# B&R Automation Studio project x20ost (part 5)

#### bnrsmartsensor.c
```c
/********************************************************************
 * COPYRIGHT -- Kontora
 ********************************************************************
 * Program: bnrmain
 * File: bnrlsens.c
 * Author: Abramenya
 * Created: January 19, 2009
 *******************************************************************/

#include "bnrsmartsensor.h"
#if MYSYSTEM_ID != 5
#ifdef _DEFAULT_INCLUDES
 #include <AsDefault.h>
#endif
extern BYTE *chSensType[];
extern BYTE *chParType[];
#ifdef WIN32
void LCPIDpara(LCPIDpara_typ *pPara){}
void LCPID(LCPID_typ *pPid){};
void LCCounter(LCCounter_typ *pCounder){};
#endif
_GLOBAL LCPIDpara_typ lParaTyp;
void CSmartSensor_InitSensor(This,PVOID pvParam)
{
    DECLARE_MULTI_OPEN(CSmartSensor,CSensor)
	SNSPARAMTABLE *pParam = (SNSPARAMTABLE*)pvParam;
	COutGate *pG = pB->m_pOutGate[0];
    pT->SetState(pT,TRUE);
	pT->m_wExtError = 0;
	pT->m_sSNSParam.enable    = pT->GetState(pT);
	pT->m_sSNSParam.enter     = pT->GetState(pT);
	pT->m_sSNSParam.Y_min     = (UINT)(pG->m_rMinRamp*pB->m_sPT.m_swMaxAcpOut);
	pT->m_sSNSParam.Y_max     = (UINT)(pG->m_rMaxRamp*pB->m_sPT.m_swMaxAcpOut);
	pT->m_sSNSParam.dY_max    = pB->m_sPT.m_rlDy;
	pT->m_sSNSParam.Kp        = pB->m_sPT.m_rlKp;
	pT->m_sSNSParam.Tn        = pB->m_sPT.m_rlTn;
	pT->m_sSNSParam.Tv        = pB->m_sPT.m_rlTv;
	pT->m_sSNSParam.Tf        = pB->m_sPT.m_rlTf;
	pT->m_sSNSParam.Kw        = pB->m_sPT.m_rlKw;
	pT->m_sSNSParam.Kfbk      = pB->m_sPT.m_rlKfbk;
	pT->m_sSNSParam.fbk_mode  = LCPID_FBK_MODE_INTERN;
	if (pB->m_sPT.m_swPidDiffMode==0)pT->m_sSNSParam.d_mode = LCPID_D_MODE_X;
	if (pB->m_sPT.m_swPidDiffMode==1)pT->m_sSNSParam.d_mode = LCPID_D_MODE_E;
	pT->m_sSNSParam.calc_mode = LCPID_CALC_MODE_FAST;
	LCPIDpara(&pT->m_sSNSParam);
	pT->m_sLCPid.enable       = pT->GetState(pT);
	pT->m_sLCPid.A            = pB->m_sPT.m_rlA;//500;
	pT->m_sLCPid.Y_man	      = pB->m_sPT.m_rlYman;
	pT->m_sLCPid.Y_fbk        = 0;
	pB->m_nInPin              = pB->m_nIniValue;
	pT->m_sLCPid.X            = pB->m_nInPin;
	pT->m_sLCPid.W            = pB->m_iPHiLimit;
	pT->m_sLCPid.Y            = pB->m_pOutGate[0]->m_wCurrOpenState;
	pB->m_nOutPin             = 0;
	pT->m_sLCPid.e            = 0;
	pT->m_sLCPid.Yi           = 0;
	pT->m_sLCPid.Yp           = 0;
	pT->m_sLCPid.Yd           = 0;
	pT->m_sLCPid.hold_I       = 0;
	if (pB->m_sPT.m_sbyMode==SNS_MD_MANU)pT->SetMode(pT,LCPID_OUT_MODE_MAN);
	if (pB->m_sPT.m_sbyMode==SNS_MD_AUTO)pT->SetMode(pT,LCPID_OUT_MODE_AUTO);
    pT->m_sLCPid.ident        = pT->m_sSNSParam.ident;
	LCPID(&pT->m_sLCPid);
	#ifdef DEB_CSmartSensor
	Info("\n(%b)CISNS::>Create SNS.:%s.:%s.Rng:[%w..%w].AlarmRng:[%w..%w]",
		&pB->m_bySensorID,
		chSensType[pB->m_bySensorType],
		chParType[pB->m_byParamType],
		&pB->m_iLoLimit,&pB->m_iHiLimit,
		&pB->m_iLoAlmLimit,&pB->m_iHiAlmLimit
	);
	#endif
}
void CSmartSensor_IncInput(This,INT16 wParam)
{
    DECLARE_MULTI_OPEN(CSmartSensor,CSensor)
    pT->m_wExtError += wParam;
	//Info("\n(%b)CSMSN::>DC(%b,%b)PR_INC::%w.",&pB->m_bySystemID,&pB->m_byDirection,&pB->m_bySensorID,&pB->m_nInPin);
}
void CSmartSensor_SetInput(This,SPIN *pValue)
{
    DECLARE_MULTI_OPEN(CSmartSensor,CSensor)
	pB->m_nInPin = pValue->iValue;
    //Info("\n(%b)CSMSN::>DC(%b,%b)PR_X::%w.",&pB->m_bySystemID,&pB->m_byDirection,&pB->m_bySensorID,&pB->m_nInPin);
}
void CSmartSensor_SetOutput(This,BYTE byNumber,SPIN *pValue)
{
	DECLARE_MULTI_OPEN(CSmartSensor,CSensor)
	COutGate *pG0 = pB->m_pOutGate[byNumber];
	pB->m_nOutPin = pValue->iValue;
	if(pG0)pG0->SetGate(pG0,pB->m_nOutPin);
}
void CSmartSensor_PreProc(This)
{
    DECLARE_MULTI_OPEN(CSmartSensor,CSensor)
	CInputGate *pI = pB->m_nInp;
	if(pB->m_byPidMode==SDIR)pB->m_nInPin = pI->GetInput(pI); else
	if(pB->m_byPidMode==SINV)pB->m_nInPin = pB->m_nAcpMax-pI->GetInput(pI);
	if(pB->m_sPT.m_sbyMode==SNS_MD_LOOP) pB->m_nInPin += pT->m_wExtError;
}
_GLOBAL LCPID_typ lPtyp;
void CSmartSensor_Processing(This)
{
    DECLARE_MULTI_OPEN(CSmartSensor,CSensor)
    #ifndef WIN32
	#ifdef MY_MODEL
	REAL rRes,rOut;
	#endif
	LCCounter(&pT->m_sCounter);
	pT->m_sLCPid.W        = pB->m_iPHiLimit;
	pT->m_sLCPid.X        = pB->m_nInPin;
	pT->m_sLCPid.basetime = pT->m_sCounter.mscnt;
	LCPID(&pT->m_sLCPid);
	#ifdef MY_MODEL
	rOut = (REAL)pT->m_sLCPid.Y;
	rRes = (rOut/378.0)-2.0;
	if((pB->m_nInPin+(INT16)rRes)>32760)pB->m_nInPin = 32760;else
	if((pB->m_nInPin+(INT16)rRes)<0)pB->m_nInPin = 0;else
	pB->m_nInPin += (INT16)rRes;
	#endif
	pB->m_nOutPin = pT->m_sLCPid.Y;
    #else
	pT->m_sLCPid.W   = pB->m_iPHiLimit;
  	pT->m_sLCPid.X   = pB->m_nInPin;
	pB->m_nOutPin    = pT->m_sLCPid.Y;
    #endif
	//pB->AddStatData(pB,pT->m_sLCPid.Y,pT->m_sLCPid.Yi,pT->m_sLCPid.Yp);
}
void CSmartSensor_PostProc(This)
{
    DECLARE_MULTI_OPEN(CSmartSensor,CSensor)
	COutGate *pG0 = pB->m_pOutGate[0];
    if(pG0)pG0->SetGate(pG0,pB->m_nOutPin);
}
void CSmartSensor_Serialize(This,BOOL byDir)
{
	DECLARE_MULTI_OPEN(CSmartSensor,CSensor)
	COutGate *pG0 = pB->m_pOutGate[0];
	if (byDir==TRUE)if(pG0)pG0->SetGate(pG0,pB->m_nOutPin);
	if (byDir==FALSE)
	{
	 pT->m_sLCPid.Y = pG0->m_wCurrOpenState;
	 pG0->StopGate(pG0);
	}
}
void CSmartSensor_RunAutomat(This)
{
    DECLARE_MULTI_OPEN(CSmartSensor,CSensor)
	BYTE i;
	COutGate *pG;
	if(pB->m_dwAutoTime++%5==0)
	{
	 pB->EventGen(pB);
	 for (i=0;i<pB->m_byAmOutGate;i++){pG = pB->m_pOutGate[i];pG->RunGate(pG);}
	}
}
void CSmartSensor_CaptureData(This)
{
	DECLARE_MULTI_OPEN(CSmartSensor,CSensor)
	COutGate *pG0 = pB->m_pOutGate[0];
    pB->OpenGate(pB);
	pB->AddData(pB,(DINT)pB->m_nInPin);
	pB->AddData(pB,(DINT)pT->m_sLCPid.W);
	pB->AddData(pB,(DINT)(pG0->GetGate(pG0)));
	pB->AddData(pB,pT->m_sLCPid.e);
	pB->AddData(pB,pT->m_sLCPid.Yi);
	pB->AddData(pB,pT->m_sLCPid.Yp);
	pB->AddData(pB,pT->m_sLCPid.Yd);
	pB->CloseGate(pB);
}
USINT CSmartSensor_GetMode(This)
{
    DECLARE_MULTI_OPEN(CSmartSensor,CSensor)
	return pT->m_sLCPid.out_mode;
}
void CSmartSensor_SetMode(This,USINT uMode)
{
    DECLARE_MULTI_OPEN(CSmartSensor,CSensor)
	pT->m_sLCPid.out_mode = uMode;
}
BOOL CSmartSensor_GetState(This)
{
    DECLARE_MULTI_OPEN(CSmartSensor,CSensor)
	return pT->m_blState;
}
void CSmartSensor_SetState(This,BOOL blBool)
{
    DECLARE_MULTI_OPEN(CSmartSensor,CSensor)
	pT->m_sSNSParam.enable    = blBool;
	pT->m_sSNSParam.enter     = blBool;
	pT->m_sLCPid.enable       = blBool;
	pT->m_blState             = blBool;
	LCPIDpara(&pT->m_sSNSParam);
}
//_GLOBAL REAL rKP;
//_GLOBAL INT  i16Param;
void CSmartSensor_EventHandler(This,SMESSAGE *pMsg)
{
    DECLARE_MULTI_OPEN(CSmartSensor,CSensor)
	SPIN nPin;
	REAL rlParam;
	INT16 wParam;
	BYTE byLen,byInitType,byPType,byPLen,*pR=(BYTE*)&rlParam;
	switch(pMsg->m_sbyType)
	{
      case EV_SMSNS_SET_PARAM_REQ:
		   byLen      = pMsg->m_sbyInfo[0];
		   byInitType = pMsg->m_sbyInfo[1];
		   byPType    = pMsg->m_sbyInfo[2];
		   byPLen     = pMsg->m_sbyInfo[3];
           #ifdef DEB_CSmartSensor
 		   //Info("\n(%b)CSMSN::>DC(%b,%b)SSP:%M.",&pB->m_bySystemID,&pB->m_byDirection,&pB->m_bySensorID,(BYTE*)pMsg);
           #endif
		   if(byInitType==SNS_SENS_OUT)
		   {
			 switch(byPType)
			 {
			  case PR_OMIN:
				   rlParam = pB->GetRealParam(pT,&pMsg->m_sbyInfo[4]);
				   pT->m_sSNSParam.Y_min = (UINT)(rlParam*pB->m_sPT.m_swMaxAcpOut);
				   LCPIDpara(&pT->m_sSNSParam);
			  break;
			  case PR_OMAX:
				   rlParam = pB->GetRealParam(pB,&pMsg->m_sbyInfo[4]);
				   pT->m_sSNSParam.Y_max = (UINT)(rlParam*pB->m_sPT.m_swMaxAcpOut);
				   LCPIDpara(&pT->m_sSNSParam);
			  break;
			  default:
			  break;
			 }
		   }
		   if(byInitType==SNS_PARA_INI)
		   {
		    switch(byPType)
			{
			 case PR_Y_max:
				  pT->m_sSNSParam.Y_max  = pB->GetWordParam(pB,&pMsg->m_sbyInfo[4]);
				  pB->m_sGT.wHiLimit     = pT->m_sSNSParam.Y_max;
                  pB->m_pOutGate[0]->SetHiLimit(pB->m_pOutGate[0],pB->m_sGT.wHiLimit);
			 break;
			 case PR_Y_min:
				  pT->m_sSNSParam.Y_min  = pB->GetWordParam(pB,&pMsg->m_sbyInfo[4]);
			 break;
			 case PR_dY_max:
				  pT->m_sSNSParam.dY_max = pB->GetRealParam(pB,&pMsg->m_sbyInfo[4]);
				  pB->m_sPT.m_rlDy       = pT->m_sSNSParam.dY_max;
			 break;
			 case PR_Kp:
				  pT->m_sSNSParam.Kp     = pB->GetRealParam(pB,&pMsg->m_sbyInfo[4]);
				  pB->m_sPT.m_rlKp       = pT->m_sSNSParam.Kp;
			 break;
			 case PR_Tn:
				  pT->m_sSNSParam.Tn     = pB->GetRealParam(pB,&pMsg->m_sbyInfo[4]);
				  pB->m_sPT.m_rlTn       = pT->m_sSNSParam.Tn;
			 break;
			 case PR_Tv:
				  pT->m_sSNSParam.Tv     = pB->GetRealParam(pB,&pMsg->m_sbyInfo[4]);
				  pB->m_sPT.m_rlTv       = pT->m_sSNSParam.Tv;
			 break;
			 case PR_Tf:
				  pT->m_sSNSParam.Tf     = pB->GetRealParam(pB,&pMsg->m_sbyInfo[4]);
				  pB->m_sPT.m_rlTf       = pT->m_sSNSParam.Tf;
			 break;
			 case PR_Kw:
				  pT->m_sSNSParam.Kw     = pB->GetRealParam(pB,&pMsg->m_sbyInfo[4]);
				  pB->m_sPT.m_rlKw       = pT->m_sSNSParam.Kw;
			 break;
			 case PR_Kfbk:
				  pT->m_sSNSParam.Kfbk   = pB->GetRealParam(pB,&pMsg->m_sbyInfo[4]);
				  pB->m_sPT.m_rlKfbk     = pT->m_sSNSParam.Kfbk;
			 break;
			 case PR_PrEn:
				  pB->m_sPT.m_swPidDiffMode = 0;
				  pT->m_sSNSParam.enable = (BOOL)pMsg->m_sbyInfo[4];
				  pB->m_sPT.m_swPidDiffMode = pT->m_sSNSParam.enable;
				  if (pB->m_sPT.m_swPidDiffMode==0)pT->m_sSNSParam.d_mode = LCPID_D_MODE_X;
				  if (pB->m_sPT.m_swPidDiffMode==1)pT->m_sSNSParam.d_mode = LCPID_D_MODE_E;
				  #ifdef DEB_CSmartSensor
				  Info("\n(%b)CSMSN::>DC(%b,%b)PR_PrEn.",&pB->m_bySystemID,&pB->m_byDirection,&pB->m_bySensorID);
				  #endif
			 break;
			 default:
			 break;
			}
		    LCPIDpara(&pT->m_sSNSParam);
		   }
		   if((byInitType==SNS_PIDC_INI)||(byInitType==SNS_SENS_INI))
		   {
			switch(byPType)
			{
			 case PR_W:
				  wParam = pB->GetWordParam(pB,&pMsg->m_sbyInfo[4]);
				  if(pB->m_byPidMode==SINV) wParam = pB->m_nAcpMax-wParam;
				  pB->m_sPT.m_swHiOper = pB->AcpToReal(pB,wParam);
   			      pT->m_sLCPid.W = wParam;
				  pB->SetHiLimit(pB,wParam);
			 break;
			 case PR_X:
				  nPin.iValue = pB->GetWordParam(pB,&pMsg->m_sbyInfo[4]);
				  pT->m_sLCPid.X = nPin.iValue;
    			  pT->SetInput(pT,&nPin);
			 break;
			 case PR_A:
				  pT->m_sLCPid.A  = pB->GetWordParam(pB,&pMsg->m_sbyInfo[4]);
				  pB->m_sPT.m_rlA = pT->m_sLCPid.A;
			 break;
			 case PR_Y_man:
				  pT->m_sLCPid.Y_man = pB->GetWordParam(pB,&pMsg->m_sbyInfo[4]);
				  pB->m_sPT.m_rlYman = pT->m_sLCPid.Y_man;
			 break;
			 case PR_out_mode:
			      if(pMsg->m_sbyInfo[4]==0)
				  {
				   #ifdef DEB_CSmartSensor
				   Info("\n(%b)CSMSN::>DC(%b,%b)SNS_MD_MANU.",&pB->m_bySystemID,&pB->m_byDirection,&pB->m_bySensorID);
				   #endif
				  }
			      if(pMsg->m_sbyInfo[4]==1)
				  {
				   pT->m_sLCPid.out_mode = LCPID_OUT_MODE_AUTO;
				   #ifdef DEB_CSmartSensor
				   Info("\n(%b)CSMSN::>DC(%b,%b)SNS_MD_AUTO.",&pB->m_bySystemID,&pB->m_byDirection,&pB->m_bySensorID);
				   #endif
				  }
			      if(pMsg->m_sbyInfo[4]==2)
				  {
				   pT->m_sLCPid.out_mode = LCPID_OUT_MODE_AUTO;
				   #ifdef DEB_CSmartSensor
				   Info("\n(%b)CSMSN::>DC(%b,%b)SNS_MD_LOOP.",&pB->m_bySystemID,&pB->m_byDirection,&pB->m_bySensorID);
				   #endif
				  }
			 break;
			 case PR_PidEn:
				  pT->m_sLCPid.enable   = (BOOL)pMsg->m_sbyInfo[4];
				  #ifdef DEB_CSmartSensor
				  Info("\n(%b)CSMSN::>DC(%b,%b)PR_PidEn.",&pB->m_bySystemID,&pB->m_byDirection,&pB->m_bySensorID);
				  #endif
			 break;
			 default:
			 break;
			}
			LCPID(&pT->m_sLCPid);
		   }
  	  break;
	  default:
	  break;
	};
}
void CSmartSensor_GetParam(This,BYTE byOwner)
{
    DECLARE_MULTI_OPEN(CSmartSensor,CSensor)
	SHMESSAGE m_sMsg;
	BYTE *pP = &m_sMsg.m_sbyInfo[1];
	SPIDPARAM sP;
	INT nSS = sizeof(SPIDPARAM);
    m_sMsg.m_sbyFrom      = MDL_DIRMD;
    m_sMsg.m_sbyFor       = byOwner;
    m_sMsg.m_sbyIntType   = DEV_ARM_PORT_TCP;
    m_sMsg.m_sbyType      = EV_SENSR_GET_PDPARAM_IND;
    m_sMsg.m_sbyServerID  = pB->m_bySystemID;
    m_sMsg.m_sbyDirection = pB->m_byDirection;
	m_sMsg.m_sbySensor  = pB->m_bySensorID;
    sP.Kp     = pB->GetRealParam(pB,(BYTE*)&pT->m_sSNSParam.Kp);
    sP.Tn     = pB->GetRealParam(pB,(BYTE*)&pT->m_sSNSParam.Tn);
    sP.Tv     = pB->GetRealParam(pB,(BYTE*)&pT->m_sSNSParam.Tv);
    sP.Tf     = pB->GetRealParam(pB,(BYTE*)&pT->m_sSNSParam.Tf);
    sP.Kw     = pB->GetRealParam(pB,(BYTE*)&pT->m_sSNSParam.Kw);
	sP.Kfbk   = pB->GetRealParam(pB,(BYTE*)&pT->m_sSNSParam.Kfbk);
	sP.Y_max  = pB->GetWordParam(pB,(BYTE*)&pT->m_sSNSParam.Y_max);
    sP.Y_min  = pB->GetWordParam(pB,(BYTE*)&pT->m_sSNSParam.Y_min);
    sP.dY_max = pB->GetRealParam(pB,(BYTE*)&pT->m_sSNSParam.dY_max);
    sP.enable = (BYTE)pT->m_sSNSParam.enable;
	pT->m_sLCPid.W = pB->m_iPHiLimit;
	sP.W      = pB->GetWordParam(pB,(BYTE*)&pT->m_sLCPid.W);
	sP.X      = pB->GetWordParam(pB,(BYTE*)&pT->m_sLCPid.X);
	sP.A      = pB->GetWordParam(pB,(BYTE*)&pT->m_sLCPid.A);
	sP.Y_man  = pB->GetWordParam(pB,(BYTE*)&pT->m_sLCPid.Y_man);
    if(pT->m_sLCPid.out_mode == LCPID_OUT_MODE_MAN) sP.out_mode = 0;
	if(pT->m_sLCPid.out_mode == LCPID_OUT_MODE_AUTO)sP.out_mode = 1;
	sP.enabled = (BYTE)pT->m_sLCPid.enable;
	m_sMsg.m_sbyInfo[0] = 1+ sizeof(SPIDPARAM);
	memcpy(&m_sMsg.m_sbyInfo[1],&sP,sizeof(SPIDPARAM));
    m_sMsg.m_swLen = 9 + m_sMsg.m_sbyInfo[0];
	#ifdef DEB_CSmartSensor
	Info("\n(%b)CSMSN::>DC(%b,%b)SFF:%M.",&pB->m_bySystemID,&pB->m_byDirection,&pB->m_bySensorID,(BYTE*)&m_sMsg);
	#endif
    FPUT(DEV_ARMOT_BOX_ID,(BYTE*)&m_sMsg.m_swLen);
}
DWORD CSmartSensor_MotToInt(This,DWORD dwData)
{
    DECLARE_MULTI_OPEN(CSmartSensor,CSensor)
	DWORD dwValue;
	BYTE *pTR = (BYTE*)&dwValue;
	BYTE *pSR = (BYTE*)&dwData;
    #ifndef WIN32
	pTR[3] = pSR[0];
	pTR[2] = pSR[1];
	pTR[1] = pSR[2];
	pTR[0] = pSR[3];
    #else
	memcpy(pTR,pSR,4);
    #endif
	return dwValue;
}
void CSmartSensor_CSmartSensor(This)
{
    DECLARE_MULTI_OPEN(CSmartSensor,CSensor)
	DECLARE_REGISTRATION(CSmartSensor,SetMode)
	DECLARE_REGISTRATION(CSmartSensor,SetState)
	DECLARE_REGISTRATION(CSmartSensor,GetState)
	DECLARE_REGISTRATION(CSmartSensor,MotToInt)
	DECLARE_VIRTUAL_FUNC(CSmartSensor,EventHandler)
	DECLARE_VIRTUAL_FUNC(CSmartSensor,SetInput)
	DECLARE_VIRTUAL_FUNC(CSmartSensor,SetOutput)
	DECLARE_VIRTUAL_FUNC(CSmartSensor,InitSensor)
	DECLARE_VIRTUAL_FUNC(CSmartSensor,PreProc)
	DECLARE_VIRTUAL_FUNC(CSmartSensor,Processing)
	DECLARE_VIRTUAL_FUNC(CSmartSensor,PostProc)
	DECLARE_VIRTUAL_FUNC(CSmartSensor,CaptureData)
	DECLARE_VIRTUAL_FUNC(CSmartSensor,GetParam)
	DECLARE_VIRTUAL_FUNC(CSmartSensor,IncInput)
	DECLARE_VIRTUAL_FUNC(CSmartSensor,RunAutomat)
	DECLARE_VIRTUAL_FUNC(CSmartSensor,Serialize)
}
void CSmartSensor_DCSmartSensor(This)
{
	DECLARE_MULTI_OPEN(CSmartSensor,CSensor)
	DestroyObjectB(CSensor,pB);
}
DECLARE_MULTI_CREATE(CSmartSensor,CSensor)
#endif
```

#### bnrsystemtimer.c
```c
/********************************************************************
 * COPYRIGHT -- Kontora
 ********************************************************************
 * Program: bnrmain
 * File: bnrlsens.c
 * Author: Abramenya
 * Created: January 19, 2009
 *******************************************************************/

#include "bnrsystemtimer.h"
#ifdef _DEFAULT_INCLUDES
 #include <AsDefault.h>
#endif
void CSystemTimer_RunTimer(This)
{
     DECLARE_SINGLE_OPEN(CSystemTimer)
	 if(pT->m_blTimerState==TRUE)
	 {
	  //Info("\nTime[%w]",&pT->m_dwTime);
      if (pT->m_dwTime--==0)
	  {
		 //Info("\nTime[%w]",&pT->m_dwTime);
         pT->DoAction(pC);
		 pT->m_dwTime = 0;
		 pT->m_blTimerState = FALSE;
		 return;
	  }
	 }
}
void CSystemTimer_DoAction(This)
{
     DECLARE_SINGLE_OPEN(CSystemTimer)
}
void CSystemTimer_OfTimer(This)
{
     DECLARE_SINGLE_OPEN(CSystemTimer)
	 pT->m_blTimerState = FALSE;
     pT->m_dwTime = 0;
}
void CSystemTimer_OnTimer(This,DWORD dwTime)
{
     DECLARE_SINGLE_OPEN(CSystemTimer)
	 pT->m_blTimerState = TRUE;
     pT->m_dwTime = dwTime;
}
void CSystemTimer_SetTimerID(This,BYTE byTimerID)
{
     DECLARE_SINGLE_OPEN(CSystemTimer)
	 pT->m_byTimerID = byTimerID;
}
void CSystemTimer_CSystemTimer(This)
{
     DECLARE_SINGLE_OPEN(CSystemTimer)
	 DECLARE_REGISTRATION(CSystemTimer,RunTimer)
	 DECLARE_REGISTRATION(CSystemTimer,OnTimer)
	 DECLARE_REGISTRATION(CSystemTimer,OfTimer)
	 DECLARE_REGISTRATION(CSystemTimer,DoAction)
	 DECLARE_REGISTRATION(CSystemTimer,SetTimerID)
	 pT->m_dwTime = 0;
	 pT->m_blTimerState = FALSE;
	 FCTIMER(pT);
}
void CSystemTimer_DCSystemTimer(This)
{
	 DECLARE_SINGLE_OPEN(CSystemTimer)
	 FDTIMER(pT);
}
DECLARE_SINGLE_CREATE(CSystemTimer)
```

#### bnrtelecontrol.c
```c
/********************************************************************
 * COPYRIGHT -- Kontora
 ********************************************************************
 * Program: bnrmain
 * File: bnrlsens.c
 * Author: Abramenya
 * Created: January 19, 2009
 *******************************************************************/

#include "bnrtelecontrol.h"
#ifdef _DEFAULT_INCLUDES
#include <AsDefault.h>
#endif
void CTeleControl_InitTCHN(This,PVOID psTable)
{
    DECLARE_MULTI_OPEN(CTeleControl,CTeleSensor)
	//BYTE i;
	pT->pP       = (STUPARAM*)psTable;
	pT->m_pbOT   = (BOOL*)pB->m_pvValue;
	pB->m_byType = REG_SOFTU_ADDR;
	pT->m_byStPulce  = FALSE;
	//pB->SaveChange(pB,EV_INI_CH,*pT->m_pbOT);
	//for(i=0;i<5;i++) pB->SaveChange(pB,EV_1T0_CH,i);
	//pT->m_bySetPulce = pT->pP->byCSetPulce;
    #ifdef DEB_CTeleControl
	//Info("\n(%b)CTLCT::>Create CTeleControl.",&pB->m_byID);
    #endif
}
void CTeleControl_PreProc(This)
{
    DECLARE_MULTI_OPEN(CTeleControl,CTeleSensor)
}
_GLOBAL INT nTCCH;
void CTeleControl_Processing(This)
{
	DECLARE_MULTI_OPEN(CTeleControl,CTeleSensor)
	if (pB->m_byID==5)	nTCCH++;
	if(pT->pP->byState==EN_OPEN)
	{
	 if(pT->m_byStPulce==TRUE)
	 {
	 if (--pT->m_bySetPulce==0)
	 {
	   if(*pT->m_pbOT==FALSE)
	   {
	   *pT->m_pbOT = TRUE;
	   pB->SaveChange(pB,EV_0T1_ST,1,FALSE);
	   }else
	   if(*pT->m_pbOT==TRUE )
	   {
	   *pT->m_pbOT = FALSE;
	   pB->SaveChange(pB,EV_1T0_ST,0,FALSE);
	   }
       #ifdef DEB_CTeleControl
	   Info("\n(%b)CTLCT::>SetPulce::STOP.",&pB->m_byID);
       #endif
	   pT->m_byStPulce  = FALSE;
	 }
	 }
	 pT->pP->byParam = *pT->m_pbOT;
	}
}
void CTeleControl_PostProc(This)
{
	DECLARE_MULTI_OPEN(CTeleControl,CTeleSensor)
}
void CTeleControl_SetPulce(This)
{
    DECLARE_MULTI_OPEN(CTeleControl,CTeleSensor)
	if(pT->pP->byState==EN_OPEN)
	{
	 pT->m_bySetPulce = pT->pP->byCSetPulce;
	 pT->m_byStPulce  = TRUE;
	 if (pT->pP->byPulceType==EN_DIRECT)
	 {
	  *pT->m_pbOT = TRUE;
	  pB->SaveChange(pB,EV_0T1_ST,1,FALSE);
	 }
	 if (pT->pP->byPulceType==EN_INVERT)
	 {
	  *pT->m_pbOT = FALSE;
	  pB->SaveChange(pB,EV_1T0_ST,0,FALSE);
	 }
	 #ifdef DEB_CTeleControl
	 Info("\n(%b)CTLCT::>SetPulce::START.",&pB->m_byID);
     #endif
	}
}
void CTeleControl_SetInPinEvent(This)
{
    DECLARE_MULTI_OPEN(CTeleControl,CTeleSensor)
	pB->SavePinState(pB,EV_INI_CH,*pT->m_pbOT);
}
void CTeleControl_SaveAlarmPin(This)
{
	DECLARE_MULTI_OPEN(CTeleControl,CTeleSensor)
	pB->SavePinState(pB,EV_ALP_CH,(WORD)pT->pP->byAlmState);
}
void CTeleControl_SendObsrveMsg(This)
{
    DECLARE_MULTI_OPEN(CTeleControl,CTeleSensor)
    SKPEVENT sEV;
	sEV.wLen    = sizeof(SKPEVENT);
	sEV.byType  = pB->m_byType;
    sEV.byCause = EV_CHK_CH;
	sEV.byAddr  = pB->m_byID;
	sEV.wValue  = (WORD)*pT->m_pbOT;
	GetCurTime(&sEV.sTime);
    pB->SendBroadcast(pB,&sEV);
}
BOOL CTeleControl_EventHandler(This,SMESSAGE *pMsg)
{
    DECLARE_MULTI_OPEN(CTeleControl,CTeleSensor)
	BYTE byParamType = pMsg->m_sbyInfo[3];
    #ifdef DEB_CTeleControl
	Info("\n(%b)CTLCT::>INPT::%M",&pB->m_byID,pMsg);
    #endif
	switch(pMsg->m_sbyFor)
	{
	  case DIR_101TOKP:
		   switch(pMsg->m_sbyType)
		   {
		    case PL_DATA_IND:
				 switch(byParamType)
				 {
				   case EN_STT_PULCE:
					    pT->SetPulce(pT);
				   break;
				   case EN_STT_SIGN:
					   //pT->SetPulce(pT,pT->pP->byPulceType);
				   break;
				   default:
				   break;
				 }

		    break;
			default:
            break;
		   }
      break;
	  case DIR_101MD:
	  break;
	  default:
	  break;
	}
	return TRUE;
}
void CTeleControl_CTeleControl(This)
{
    DECLARE_MULTI_OPEN(CTeleControl,CTeleSensor)
	DECLARE_REGISTRATION(CTeleControl,SetPulce)
	DECLARE_VIRTUAL_FUNC(CTeleControl,SetInPinEvent)
	DECLARE_VIRTUAL_FUNC(CTeleControl,InitTCHN)
	DECLARE_VIRTUAL_FUNC(CTeleControl,PreProc)
	DECLARE_VIRTUAL_FUNC(CTeleControl,Processing)
	DECLARE_VIRTUAL_FUNC(CTeleControl,PostProc)
	DECLARE_VIRTUAL_FUNC(CTeleControl,EventHandler)
	DECLARE_VIRTUAL_FUNC(CTeleControl,SaveAlarmPin)
	DECLARE_VIRTUAL_FUNC(CTeleControl,SendObsrveMsg)
}
void CTeleControl_DCTeleControl(This)
{
	DECLARE_MULTI_OPEN(CTeleControl,CTeleSensor)
}
DECLARE_MULTI_CREATE(CTeleControl,CTeleSensor)
```

#### bnrteleind.c
```c
/********************************************************************
 * COPYRIGHT -- Kontora
 ********************************************************************
 * Program: bnrmain
 * File: bnrlsens.c
 * Author: Abramenya
 * Created: January 19, 2009
 *******************************************************************/

#include "bnrteleind.h"
#include "bnrmain.h"
#ifdef _DEFAULT_INCLUDES
#include <AsDefault.h>
#endif
extern UINT *uipValueAI2[];
void CTeleInd_InitTCHN(This,PVOID psTable)
{
    DECLARE_MULTI_OPEN(CTeleInd,CTeleSensor)
	//BYTE i;
	pT->pP = (STIPARAM*)psTable;
	pT->m_pnIN = (WORD*)pB->m_pvValue;

	pT->m_byRemTimer   = pT->pP->byDrTimer;
	pT->m_blTmRemState = FALSE;

	pT->m_bySetTimer   = pT->pP->byDrTimer;
	pT->m_blTmSetState = FALSE;

	pT->m_blChState    = pT->pP->byDrTimer;
	pT->m_byChTimer    = FALSE;

	pT->m_byErEventCh  = EV_CHG_PR;
	pT->m_byErEventHi  = EV_CHG_PR;
	pT->m_byErEventLo  = EV_CHG_PR;
	pB->m_byType       = REG_SOFTI_ADDR;
	//pB->SaveChange(pB,EV_INI_CH,*pT->m_pnIN);
    pT->InitMeter(pT);
	//for(i=0;i<5;i++) pB->SaveChange(pB,pT->m_byEvent,i);
    #ifdef DEB_CTeleInd
	//Info("\n(%b)CTIMD::>Create CTeleInd:",&pB->m_byID);
    #endif
}
void CTeleInd_InitMeter(This)
{
    DECLARE_MULTI_OPEN(CTeleInd,CTeleSensor)
	WORD wIN = *pT->m_pnIN;
	if(wIN>=pT->pP->wHiLimit)
	{
	 pT->m_blSHIL   = TRUE;
	 pT->m_blRHIL   = FALSE;
	 pT->m_blSLOL   = FALSE;
	 pT->m_blRLOL   = TRUE;
	}
	if(wIN<=pT->pP->wLoLimit)
	{
	 pT->m_blSLOL   = TRUE;
	 pT->m_blRLOL   = FALSE;
	 pT->m_blSHIL   = FALSE;
	 pT->m_blRHIL   = TRUE;
	}
	if((wIN<=pT->pP->wHiGister)&&(wIN>=pT->pP->wLoGister))
	{
	 pT->m_blSHIL   = FALSE;
	 pT->m_blRHIL   = TRUE;
	 pT->m_blSLOL   = FALSE;
	 pT->m_blRLOL   = TRUE;
	}
	pT->m_wOldIN = wIN;
}
void CTeleInd_PreProc(This)
{
    DECLARE_MULTI_OPEN(CTeleInd,CTeleSensor)
	BOOL res = FALSE;

	if(pT->m_blTmSetState==TRUE)
	{
	 if (--pT->m_bySetTimer==0)
	 {
	  if((pT->pP->byPriority==PRI_HI)&&(pT->m_byErEventHi==EV_SET_HI))res = TRUE;
	  pB->SaveChange(pB,pT->m_byErEventHi,*pT->m_pnIN,res);
	  pT->m_blTmSetState = FALSE;
	 }
	}
	res = FALSE;

	if(pT->m_blTmRemState==TRUE)
	{
	 if (--pT->m_byRemTimer==0)
	 {
	  if((pT->pP->byPriority==PRI_HI)&&(pT->m_byErEventLo==EV_SET_LO))res = TRUE;
	  pB->SaveChange(pB,pT->m_byErEventLo,*pT->m_pnIN,res);
	  pT->m_blTmRemState = FALSE;
	 }
	}
	res = FALSE;

	if(pT->m_blChState==TRUE)
	{
	 if (--pT->m_byChTimer==0)
	 {
	  //Info("\n(%b)CTIMD::>TI:%w",&pB->m_byID,pT->m_pnIN);
	  if(pT->pP->byPriority==PRI_HI)res = TRUE;
	  pB->SaveChange(pB,pT->m_byErEventCh,*pT->m_pnIN,FALSE);
	  pT->m_blChState = FALSE;
	 }
	}

}
void CTeleInd_Processing(This)
{
	DECLARE_MULTI_OPEN(CTeleInd,CTeleSensor)
	if(pT->pP->byState==EN_OPEN)
	{
  	 pT->CheckTI(pT);
     pT->pP->wParam = *pT->m_pnIN;
	}
}
void CTeleInd_PostProc(This)
{
	DECLARE_MULTI_OPEN(CTeleInd,CTeleSensor)
}
_GLOBAL INT nTICH;
WORD CTeleInd_CheckTI(This)
{
    DECLARE_MULTI_OPEN(CTeleInd,CTeleSensor)
	WORD res;
	WORD wIN = *pT->m_pnIN;
	WORD wHI =  pT->pP->wHiLimit;
	WORD wLO =  pT->pP->wLoLimit;
	WORD wHG =  pT->pP->wHiGister;
	WORD wLG =  pT->pP->wLoGister;
	//Deviation Section
	if(abs(wIN-pT->m_wOldIN)>pT->pP->wEvPercent)
	{
		pT->SetChandgeTimer(pT,EV_CHG_PR);
		pT->m_wOldIN = wIN;
	}
	//Hi Section
	//if (pB->m_byID==0)
	//if ((++nTICH % 20)==0)Info("\n(__)IN:%w HI:%w HG:%w LG:%w LO:%w BRLO:%b BSLO:%b",&wIN,&wHI,&wHG,&wLG,&wLO,&pT->m_blRLOL,&pT->m_blSLOL);
	if(wIN>=wHI)
	{
	  pT->SetEventHi(pT,&pT->m_blSHIL,&pT->m_blRHIL,EV_SET_HI);
	}
	//if((wIN<wHG)&&(wIN>wLG))
	if(wIN<wHG)
	{
	  pT->SetEventHi(pT,&pT->m_blRHIL,&pT->m_blSHIL,EV_REM_HI);
	}
	//if((wIN>wLG)&&(wIN<wHG))
	if(wIN>wLG)
	{
	  pT->SetEventLo(pT,&pT->m_blRLOL,&pT->m_blSLOL,EV_REM_LO);
	}
	if(wIN<wLO)
	{
	  pT->SetEventLo(pT,&pT->m_blSLOL,&pT->m_blRLOL,EV_SET_LO);
	}
	return res=wIN;
}
void CTeleInd_SetEventHi(This,BOOL *bl0,BOOL *bl1,BYTE byEvent)
{
    DECLARE_MULTI_OPEN(CTeleInd,CTeleSensor)
	if (*bl0 == FALSE)
	{
	 pT->SetEventTimerHi(pT,byEvent);
     *bl0 = TRUE;
     *bl1 = FALSE;
	}
}
void CTeleInd_SetEventLo(This,BOOL *bl0,BOOL *bl1,BYTE byEvent)
{
    DECLARE_MULTI_OPEN(CTeleInd,CTeleSensor)
	if (*bl0 == FALSE)
	{
	 pT->SetEventTimerLo(pT,byEvent);
     *bl0 = TRUE;
     *bl1 = FALSE;
	}
}
void CTeleInd_SetEventEv(This,BOOL *bl0,BOOL *bl1,BYTE byEvent)
{
    DECLARE_MULTI_OPEN(CTeleInd,CTeleSensor)
	if (*bl0 == FALSE)
	{
	 //pT->SetEventTimer(pT,byEvent);
	 pT->m_byErEventCh = byEvent;
	 pB->SaveChange(pB,pT->m_byErEventCh,*pT->m_pnIN,FALSE);
     *bl0 = TRUE;
     *bl1 = FALSE;
	}
}
void CTeleInd_SetEventTimerHi(This,BYTE byEvent)
{
	DECLARE_MULTI_OPEN(CTeleInd,CTeleSensor)
	pT->m_blTmSetState = TRUE;
	pT->m_bySetTimer   = pT->pP->byDrTimer;
	pT->m_byErEventHi  = byEvent;
}
void CTeleInd_SetEventTimerLo(This,BYTE byEvent)
{
	DECLARE_MULTI_OPEN(CTeleInd,CTeleSensor)
	pT->m_blTmRemState = TRUE;
	pT->m_byRemTimer   = pT->pP->byDrTimer;
	pT->m_byErEventLo  = byEvent;
}
void CTeleInd_SetChandgeTimer(This,BYTE byEvent)
{
	DECLARE_MULTI_OPEN(CTeleInd,CTeleSensor)
	pT->m_blChState    = TRUE;
	pT->m_byChTimer    = pT->pP->byDrTimer;
	pT->m_byErEventCh  = byEvent;
}
void CTeleInd_SetInPinEvent(This)
{
    DECLARE_MULTI_OPEN(CTeleInd,CTeleSensor)
	pB->SavePinState(pB,EV_INI_CH,*pT->m_pnIN);
}
void CTeleInd_SaveAlarmPin(This)
{
	DECLARE_MULTI_OPEN(CTeleInd,CTeleSensor)
	pB->SavePinState(pB,EV_ALP_CH,(WORD)pT->pP->byAlmState);
}
void CTeleInd_SendObsrveMsg(This)
{
    DECLARE_MULTI_OPEN(CTeleInd,CTeleSensor)
    SKPEVENT sEV;
	sEV.wLen    = sizeof(SKPEVENT);
	sEV.byType  = pB->m_byType;
    sEV.byCause = EV_CHK_CH;
	sEV.byAddr  = pB->m_byID;
	sEV.wValue  = (WORD)*pT->m_pnIN;
	GetCurTime(&sEV.sTime);
    pB->SendBroadcast(pB,&sEV);
}
BOOL CTeleInd_EventHandler(This,SMESSAGE *pMsg)
{
	DECLARE_MULTI_OPEN(CTeleInd,CTeleSensor)
	BYTE byParamType = pMsg->m_sbyInfo[3];
    #ifdef DEB_CTeleInd
	Info("\n(%b)CTIMD::>INPT::%M",&pB->m_byID,pMsg);
    #endif
	switch(pMsg->m_sbyFor)
	{
	  case DIR_101TOKP:
		   switch(pMsg->m_sbyType)
		   {
		    case PL_DATA_IND:
				 switch(byParamType)
				 {
				   case EN_HIL_PR:
					    //pT->m_wHiLimit  = pB->GetW(pB,&pMsg->m_sbyInfo[3]);
				   break;
				   case EN_HIG_PR:
					    //pT->m_wHiGister = pB->GetW(pB,&pMsg->m_sbyInfo[3]);
				   break;
				   case EN_LOL_PR:
					    //pT->m_wLoLimit  = pB->GetW(pB,&pMsg->m_sbyInfo[3]);
				   break;
				   case EN_LOG_PR:
					    //pT->m_wLoGister = pB->GetW(pB,&pMsg->m_sbyInfo[3]);
				   break;
				   case EN_DTM_PR:
					    //pT->m_byDrTimer = pMsg->m_sbyInfo[3];
				   break;
				   default:
				   break;
				 }
		    break;
			default:
            break;
		   }
      break;
	  case DIR_101MD:
	  break;
	  default:
	  break;
	}
	return TRUE;
}
void CTeleInd_CTeleInd(This)
{
    DECLARE_MULTI_OPEN(CTeleInd,CTeleSensor)
	DECLARE_REGISTRATION(CTeleInd,CheckTI)
	DECLARE_REGISTRATION(CTeleInd,InitMeter)
	DECLARE_REGISTRATION(CTeleInd,SetEventHi)
	DECLARE_REGISTRATION(CTeleInd,SetEventLo)
	DECLARE_REGISTRATION(CTeleInd,SetEventTimerHi)
	DECLARE_REGISTRATION(CTeleInd,SetEventTimerLo)
	DECLARE_REGISTRATION(CTeleInd,SetChandgeTimer)
	DECLARE_REGISTRATION(CTeleInd,SetEventEv)

	DECLARE_VIRTUAL_FUNC(CTeleInd,InitTCHN)
	DECLARE_VIRTUAL_FUNC(CTeleInd,PreProc)
	DECLARE_VIRTUAL_FUNC(CTeleInd,Processing)
	DECLARE_VIRTUAL_FUNC(CTeleInd,PostProc)
	DECLARE_VIRTUAL_FUNC(CTeleInd,EventHandler)
	DECLARE_VIRTUAL_FUNC(CTeleInd,SetInPinEvent)
	DECLARE_VIRTUAL_FUNC(CTeleInd,SaveAlarmPin)
	DECLARE_VIRTUAL_FUNC(CTeleInd,SendObsrveMsg)
}
void CTeleInd_DCTeleInd(This)
{
	DECLARE_MULTI_OPEN(CTeleInd,CTeleSensor)
}
DECLARE_MULTI_CREATE(CTeleInd,CTeleSensor)
```

#### bnrtelesensor.c
```c
/********************************************************************
 * COPYRIGHT -- Kontora
 ********************************************************************
 * Program: bnrmain
 * File: bnrlsens.c
 * Author: Abramenya
 * Created: January 19, 2009
 *******************************************************************/

#include "bnrtelesensor.h"
#include "bnrmain.h"
#ifdef _DEFAULT_INCLUDES
 #include <AsDefault.h>
#endif
//#include "bnrmain.h"
//#ifdef WIN32
char *STTS[]  =
{
    "EV_SET_HI",
	"EV_REM_HI",
	"EV_SET_LO",
	"EV_REM_LO",
	"EV_CHG_PR",
	"EV_0T1_CH",
	"EV_1T0_CH",
	"EV_SAL_CH",
	"EV_RAL_CH",
	"EV_0T1_ST",
	"EV_1T0_ST",
	"EV_INI_CH",
	"EV_ALP_CH",
	"EV_ALS_CH",
	"EV_DSC_CH",

};
//#endif
BYTE byIDD;
void CTeleSensor_Init(This,PVOID *psTable)
{
    DECLARE_SINGLE_OPEN(CTeleSensor)
	CSlot *pSL;
	CComputer *pCM   = pT->m_pComputer;
	STIPARAM  *pPV   = (STIPARAM*)psTable;
    pT->pP           = pPV;
	pT->m_byID       = pPV->byID;
	byIDD            = pT->m_byID;
	pSL              = pCM->GetSlot(pCM,pT->pP->bySlot);
	pT->m_pPN        = pSL->GetPin(pSL->pChld,pT->pP->byPin);
	pT->m_pvValue    = (PVOID)pT->m_pPN->GetAddrPin(pT->m_pPN->pChld);
    pT->m_pvAlValue  = (BOOL*)pT->m_pPN->m_pvAlmState;
	pT->m_blSetAlarm = FALSE;
	pT->m_byOldEvent = 0xff;
	#ifdef WIN32
    if(pPV->byType==TI)
	{
	 *((WORD*)pT->m_pvValue) = pT->m_byID;
	 pT->pP->wParam = pT->m_byID;
    }
	if(pPV->byType==TU) *((BOOL*)pT->m_pvValue) = FALSE;
	#endif
	pT->InitTCHN(pC,psTable);
}
void CTeleSensor_Switch(This)
{
   DECLARE_SINGLE_OPEN(CTeleSensor)
   CSlot *pSL;
   CComputer *pCM  = pT->m_pComputer;
   pSL             = pCM->GetSlot(pCM,pT->pP->bySlot);
   pT->m_pPN       = pSL->GetPin(pSL->pChld,pT->pP->byPin);
   pT->m_pvValue   = (PVOID)pT->m_pPN->GetAddrPin(pT->m_pPN->pChld);
   pT->m_pvAlValue = (BOOL*)pT->m_pPN->m_pvAlmState;
   pT->InitTCHN(pC,pT->pP);
}
void CTeleSensor_InitTCHN(This,SSWITCHTABLE *psTable){}
void CTeleSensor_PreProc(This){}
void CTeleSensor_Processing(This){}
void CTeleSensor_PostProc(This){}
void CTeleSensor_ObserveProc(This)
{
     DECLARE_SINGLE_OPEN(CTeleSensor)
	 pT->PreProc(pC);
	 pT->Processing(pC);
	 pT->PostProc(pC);
     if(++pT->m_byALC%20==0) pT->CheckAlarm(pT);
}
void CTeleSensor_CheckAlarm(This)
{
     DECLARE_SINGLE_OPEN(CTeleSensor)
	 if(*pT->m_pvAlValue==TRUE)
	 {
      if (pT->m_blSetAlarm==FALSE)
      {
	    pT->m_blSetAlarm = TRUE;
		pT->SaveChange(pT,EV_SAL_CH,1,TRUE);
		pT->pP->byAlmState = 1;
      }
	 }else
	 if(*pT->m_pvAlValue==FALSE)
	 {
      if (pT->m_blSetAlarm==TRUE)
      {
	   pT->m_blSetAlarm = FALSE;
	   pT->SaveChange(pT,EV_RAL_CH,0,TRUE);
	   pT->pP->byAlmState = 0;
	  }
	 }
}
BOOL CTeleSensor_EventHandler(This,SMESSAGE *pMsg)
{
	 DECLARE_SINGLE_OPEN(CTeleSensor)
	 return TRUE;
}
BOOL CTeleSensor_SaveChange(This,BYTE byEvent,WORD wValue,BOOL blAlarm)
{
    DECLARE_SINGLE_OPEN(CTeleSensor)
	SKPEVENT sEV;
	STSPARAM *pTS;STIPARAM *pTI;
	SKPPARAM *pH = pT->m_pPCT->pKpParam;
	sEV.wLen    = sizeof(SKPEVENT);
	sEV.byType  = pT->m_byType;
    sEV.byCause = byEvent;
    if((byEvent!=pT->m_byOldEvent)||(byEvent==EV_CHG_PR))
	{
	 pT->m_byOldEvent = byEvent;
	 sEV.byAddr  = pT->m_byID;
	 sEV.wValue  = wValue;
	 GetCurTime(&sEV.sTime);
     if(blAlarm)
	 {
	  #ifdef DEB_CTeleSensor
      Info("\n(%b)CTLSN::>Send Alarm[%s]:",&pT->m_byID,STTS[sEV.byCause]);
      #endif
	  pT->SendSMessage(pT,DEV_KPMDL_BOX_ID,DIR_PHTOKP,PH_CALL_REQ);
	 }
	 FPUT1(BOX_L4,(BYTE*)&sEV);
	 if((pH->byStoreMode&SBM_TIUNLOAD)&&(sEV.byType==REG_SOFTI_ADDR)) pT->SendBroadcast(pT,&sEV);
	 if((pH->byStoreMode&SBM_TSUNLOAD)&&(sEV.byType==REG_SOFTS_ADDR)) pT->SendBroadcast(pT,&sEV);
	 if((pH->byStoreMode&SBM_TUUNLOAD)&&(sEV.byType==REG_SOFTU_ADDR)) pT->SendBroadcast(pT,&sEV);
	 /*
	 Info("\n(%b)CTLSN::>Y[%b]:M[%b]:D[%b]:H[%b]:M[%b]::S[%b]::L[%b]::H[%b]:",
	 &pT->m_byID,
	 &sEV.sTime.tYear,
	 &sEV.sTime.tMonth,
	 &sEV.sTime.tDay,
	 &sEV.sTime.tHour,
	 &sEV.sTime.tMin,
	 &sEV.sTime.tSec,
	 &sEV.sTime.tMSecL,
	 &sEV.sTime.tMSecH);
	 */
	 #ifdef DEB_CTeleSensor
	 Info("\n(%b)CTLSN::>TP[%b]:AD[%b]:VL[%w]:CS[%s]:",&pT->m_byID,&sEV.byType,&sEV.byAddr,&sEV.wValue,STTS[sEV.byCause]);
     #endif
	}
	return TRUE;
}
BOOL CTeleSensor_SavePinState(This,BYTE byEvent,WORD wValue)
{
    DECLARE_SINGLE_OPEN(CTeleSensor)
	SKPEVENT sEV;
	STSPARAM *pTS;
	SHARDCOMPUTERTABLE *pH = pT->m_pPCT;
	sEV.wLen    = sizeof(SKPEVENT);
	sEV.byType  = pT->m_byType;
    sEV.byCause = byEvent;
	sEV.byAddr  = pT->m_byID;
	sEV.wValue  = wValue;
	GetCurTime(&sEV.sTime);
	FPUT1(BOX_L4_1,(BYTE*)&sEV);
	#ifdef DEB_CTeleSensor
	Info("\n(%b)CTLIN::>TP[%b]:AD[%b]:VL[%w]:CS[%s]:",&pT->m_byID,&sEV.byType,&sEV.byAddr,&sEV.wValue,STTS[sEV.byCause]);
    #endif
	return TRUE;
}
void CTeleSensor_SendSMessage(This,BYTE byBox,BYTE byFor,BYTE byType)
{
    DECLARE_SINGLE_OPEN(CTeleSensor)
    SHORTMESSAGE m_sMsg;
	m_sMsg.m_swLen        = 9;
	m_sMsg.m_sbyFrom      = DIR_PHMDL;
	m_sMsg.m_sbyFor       = byFor;
	m_sMsg.m_sbyIntType   = 0;
	m_sMsg.m_sbyServerID  = 0;
	m_sMsg.m_sbyType      = byType;
	m_sMsg.m_sbyDirection = 0;
	m_sMsg.m_sbySensor    = 0;
	FPUT(byBox,(BYTE*)&m_sMsg);
    #ifdef DEB_CTeleSensor
	Info("\n(__)CTLSN::>OUTT::%M",&m_sMsg);
    #endif
}
void CTeleSensor_SendBroadcast(This,SKPEVENT *pEV)
{
    DECLARE_SINGLE_OPEN(CTeleSensor)
	SHORTMESSAGE m_sMsg	;
	m_sMsg.m_swLen        = 9 + sizeof(SKPEVENT);
	m_sMsg.m_sbyFrom      = DIR_KPMOD;
	m_sMsg.m_sbyFor       = DIR_KPTO101;
	m_sMsg.m_sbyIntType   = 0;
	m_sMsg.m_sbyServerID  = 0;
	m_sMsg.m_sbyType      = PL_DATA_REQ;
	m_sMsg.m_sbyDirection = 0;
	m_sMsg.m_sbySensor    = 0;
	memcpy(&m_sMsg.m_sbyInfo[0],pEV,sizeof(SKPEVENT));
	FPUT(DEV_101MD_BOX_ID,(BYTE*)&m_sMsg);
}
void CTeleSensor_SetInPinEvent(This)
{
    DECLARE_SINGLE_OPEN(CTeleSensor)
}
void CTeleSensor_SaveAlarmPin(This)
{
    DECLARE_SINGLE_OPEN(CTeleSensor)
}
void CTeleSensor_SendObsrveMsg(This)
{
    DECLARE_SINGLE_OPEN(CTeleSensor)
}
void CTeleSensor_CTeleSensor(This)
{
     DECLARE_SINGLE_OPEN(CTeleSensor)
	 DECLARE_REGISTRATION(CTeleSensor,Init)
	 //DECLARE_REGISTRATION(CTeleSensor,GetW)
	 DECLARE_REGISTRATION(CTeleSensor,SendSMessage)
	 DECLARE_REGISTRATION(CTeleSensor,ObserveProc)
	 DECLARE_REGISTRATION(CTeleSensor,PreProc)
	 DECLARE_REGISTRATION(CTeleSensor,Processing)
	 DECLARE_REGISTRATION(CTeleSensor,PostProc)
	 DECLARE_REGISTRATION(CTeleSensor,EventHandler)
	 DECLARE_REGISTRATION(CTeleSensor,SaveChange)
	 DECLARE_REGISTRATION(CTeleSensor,SavePinState)
	 DECLARE_REGISTRATION(CTeleSensor,SendBroadcast)
	 DECLARE_REGISTRATION(CTeleSensor,CheckAlarm)
	 DECLARE_REGISTRATION(CTeleSensor,Switch)
	 DECLARE_REGISTRATION(CTeleSensor,SetInPinEvent)
	 DECLARE_REGISTRATION(CTeleSensor,SaveAlarmPin)
	 DECLARE_REGISTRATION(CTeleSensor,SendObsrveMsg)
}
void CTeleSensor_DCTeleSensor(This)
{
	 DECLARE_SINGLE_OPEN(CTeleSensor)
}
DECLARE_SINGLE_CREATE(CTeleSensor)
```

#### bnrtelesignal.c
```c
/********************************************************************
 * COPYRIGHT -- Kontora
 ********************************************************************
 * Program: bnrmain
 * File: bnrlsens.c
 * Author: Abramenya
 * Created: January 19, 2009
 *******************************************************************/

#include "bnrtelesignal.h"
#include "bnrmain.h"
#ifdef _DEFAULT_INCLUDES
 #include <AsDefault.h>
#endif
_GLOBAL BYTE nFSignal;
void CTeleSignal_InitTCHN(This,PVOID psTable)
{
    DECLARE_MULTI_OPEN(CTeleSignal,CTeleSensor)
	//BYTE i;
	pT->pP = (STSPARAM*)psTable;
	pT->m_pbIN = (BOOL*)pB->m_pvValue;
	pT->m_blTmSetState = FALSE;
	pT->m_blTmRemState = FALSE;
	pB->m_byType       = REG_SOFTS_ADDR;
	pT->m_blFSignal    = FALSE;
	//pB->SaveChange(pB,EV_INI_CH,*pT->m_pbIN);
	//for(i=0;i<5;i++) pB->SaveChange(pB,EV_0T1_CH,i);
    #ifdef DEB_CTeleSignal
	//Info("\n(%b)CTLSG::>Create TeleSignal.",&pB->m_byID);
    #endif
}
void CTeleSignal_PreProc(This)
{
    DECLARE_MULTI_OPEN(CTeleSignal,CTeleSensor)

}
_GLOBAL INT nTSCH;
void CTeleSignal_Processing(This)
{
	DECLARE_MULTI_OPEN(CTeleSignal,CTeleSensor)
	BYTE byState;
	if (pB->m_byID==40)	nTSCH++;
	if (pT->pP->byState==EN_OPEN)
	{
	 byState = pT->CheckTS(pT);
	 if(byState==PIN_STATE_ONN){pT->m_blTmSetState = TRUE;pT->m_blTmRemState = FALSE;pT->m_bySetPulce = pT->pP->byCSetPulce;}
	 if(byState==PIN_STATE_OFF){pT->m_blTmRemState = TRUE;pT->m_blTmSetState = FALSE;pT->m_byRemPulce = pT->pP->byCRemPulce;}
	 pT->pP->byParam = *pT->m_pbIN;
	}
}
void CTeleSignal_PostProc(This)
{
	DECLARE_MULTI_OPEN(CTeleSignal,CTeleSensor)
	BOOL res = FALSE;
	//Set Timer
	if (pT->pP->byState==EN_OPEN)
	{
	if(pT->m_blTmSetState==TRUE)
	{
	 if (--pT->m_bySetPulce==0)
	 {
	  if((pT->pP->byPriority==PRI_HI)&&((pT->pP->byAlarmMode==EN_AL_TO_AL)||(pT->pP->byAlarmMode==EN_LO_TO_HI))) res = TRUE;
	  pB->SaveChange(pB,EV_0T1_CH,1,res);
	  pT->m_blTmSetState = FALSE;
	 }
	}
    //Rem Timer
	if(pT->m_blTmRemState==TRUE)
	{
	 if (--pT->m_byRemPulce==0)
	 {
	  if((pT->pP->byPriority==PRI_HI)&&((pT->pP->byAlarmMode==EN_AL_TO_AL)||(pT->pP->byAlarmMode==EN_HI_TO_LO))) res = TRUE;
	  if( pT->m_blFSignal)pB->SaveChange(pB,EV_1T0_CH,0,res);
	  pT->m_blTmRemState = FALSE;
	  pT->m_blFSignal = TRUE;
	 }
	}
	}
}
BYTE CTeleSignal_CheckTS(This)
{
    DECLARE_MULTI_OPEN(CTeleSignal,CTeleSensor)
	return pB->m_pPN->GetState(pB->m_pPN);
}
BOOL CTeleSignal_EventHandler(This,SMESSAGE *pMsg)
{
    DECLARE_MULTI_OPEN(CTeleSignal,CTeleSensor)
    BYTE byID = pMsg->m_sbySensor;
	BYTE byParamType = pMsg->m_sbyInfo[3];
    #ifdef DEB_CTeleSignal
	Info("\n(%b)CTLSG::>INPT::%M",&pB->m_byID,pMsg);
    #endif
	switch(pMsg->m_sbyFor)
	{
	  case DIR_101TOKP:
		   switch(pMsg->m_sbyType)
		   {
		    case PL_DATA_IND:
				 //Info("\n(%b)CTLSG::>DL_DATA_IND::>%M",&pB->m_byID,pMsg);
				 switch(byParamType)
				 {
				   case EN_SET_PERIOD:
					    //pT->m_byCSetPulce = pMsg->m_sbyInfo[3];
					    //pT->m_bySetPulce  = pT->m_byCSetPulce;
				   break;
				   case EN_REM_PERIOD:
					    //pT->m_byRemPulce  = pMsg->m_sbyInfo[3];
						//pT->m_byCRemPulce = pT->m_byRemPulce;
				   break;
				   case EN_PIN_ALMODE:
                        //pT->m_byAlarmMode = pMsg->m_sbyInfo[3];
				   break;
				   default:
				   break;
				 }
		    break;
			default:
            break;
		   }
      break;
	  case DIR_101MD:
	  break;
	  default:
	  break;
	}
	return TRUE;
}
void CTeleSignal_SetInPinEvent(This)
{
    DECLARE_MULTI_OPEN(CTeleSignal,CTeleSensor)
	pB->SavePinState(pB,EV_INI_CH,*pT->m_pbIN);
}
void CTeleSignal_SaveAlarmPin(This)
{
	DECLARE_MULTI_OPEN(CTeleSignal,CTeleSensor)
	pB->SavePinState(pB,EV_ALP_CH,(WORD)pT->pP->byAlmState);
}
void CTeleSignal_SendObsrveMsg(This)
{
    DECLARE_MULTI_OPEN(CTeleSignal,CTeleSensor)
    SKPEVENT sEV;
	sEV.wLen    = sizeof(SKPEVENT);
	sEV.byType  = pB->m_byType;
    sEV.byCause = EV_CHK_CH;
	sEV.byAddr  = pB->m_byID;
	sEV.wValue  = (WORD)*pT->m_pbIN;
	GetCurTime(&sEV.sTime);
    pB->SendBroadcast(pB,&sEV);
}
void CTeleSignal_CTeleSignal(This)
{
    DECLARE_MULTI_OPEN(CTeleSignal,CTeleSensor)
	DECLARE_REGISTRATION(CTeleSignal,CheckTS)
	DECLARE_VIRTUAL_FUNC(CTeleSignal,EventHandler)
	DECLARE_VIRTUAL_FUNC(CTeleSignal,InitTCHN)
	DECLARE_VIRTUAL_FUNC(CTeleSignal,PreProc)
	DECLARE_VIRTUAL_FUNC(CTeleSignal,Processing)
	DECLARE_VIRTUAL_FUNC(CTeleSignal,PostProc)
	DECLARE_VIRTUAL_FUNC(CTeleSignal,SetInPinEvent)
	DECLARE_VIRTUAL_FUNC(CTeleSignal,SaveAlarmPin)
	DECLARE_VIRTUAL_FUNC(CTeleSignal,SendObsrveMsg)
}
void CTeleSignal_DCTeleSignal(This)
{
	DECLARE_MULTI_OPEN(CTeleSignal,CTeleSensor)
}
DECLARE_MULTI_CREATE(CTeleSignal,CTeleSensor)
```

#### multi.c
```c
/********************************************************************
 * COPYRIGHT -- Kontora
 ********************************************************************
 * Program: bnrmain
 * File: bnrlsens.c
 * Author: Abramenya
 * Created: January 19, 2009
 *******************************************************************/

#include "multi.h"
#ifdef _DEFAULT_INCLUDES
 #include <AsDefault.h>
#endif
void CMulti_CMulti(This)
{
    DECLARE_MULTI_OPEN(CMulti,CSingle)
}
void CMulti_DCMulti(This)
{
	DECLARE_MULTI_OPEN(CMulti,CSingle)
}
DECLARE_MULTI_CREATE(CMulti,CSingle)
```

#### bnradmin.h
```c
/********************************************************************
 * COPYRIGHT -- Kontora
 ********************************************************************
 * Program: bnrmain
 * File: bnraninput.h
 * Author: Abramenya
 * Created: January 19, 2009
 *******************************************************************/

#ifndef __ADMIN_H__
#define __ADMIN_H__
#include "typedefs.h"
#include "bnrcyclicsystem.h"
#include "bnrmytimer.h"
#include "bnrmessage.h"
#include "bnrpob.h"
#define MAX_COMMAND_LENGTH 4
enum _tagSystemState
{
	 SYS_ST00_NULL=0,
	 SYS_ST01_DISC,
	 SYS_ST02_CONN,
	 SYS_ST03_WAIT_CONF,
	 SYS_ST04_SYST_READY,
	 SYS_ST05_WAIT_READY,
};
Class CAdmin
{
	 void (*CCAdmin)(This);
	 void (*DCAdmin)(This);
Public
     void (*Init)(This);
     BOOL (*SendMessage)(This,BYTE byBox,BYTE byFor,BYTE byType,BYTE byDir,BYTE bySens);
	 void (*PreCommHandler)(This,SMESSAGE *pMsg);
	 void (*HandCommHandler)(This,DWORD b_lCode,BYTE ps,BYTE *pbyBuffer,BYTE byLength);
	 void (*SetSystemID)(This,BYTE);
	 void (*SetState)(This,BYTE);
	 BYTE (*GetState)(This);
	 BOOL (*AdminAutomat)(This,SMESSAGE*);
	 void (*DevVersion)(This);
	 Virtual BOOL (*EventHandler)(This,SMESSAGE *pMsg);
     Virtual void (*CyclicProc)(This);
Private
     BYTE m_bySystemState;
     //SMESSAGE m_sMsg;
	 CMTimer m_pTAskConfig;
	 CMTimer m_pTSendState;
	 BOOL m_blArmState;
	 BYTE m_bySystemID;
	 DECLARE_IMPLEMENT_BASE(CCyclicSystem)
}
DECLARE_DEFINITION(CAdmin)
#endif
```

#### bnraninput.h
```c
/********************************************************************
 * COPYRIGHT -- Kontora
 ********************************************************************
 * Program: bnrmain
 * File: bnraninput.h
 * Author: Abramenya
 * Created: January 19, 2009
 *******************************************************************/

#ifndef __ANINPUT_H__
#define __ANINPUT_H__
#include "typedefs.h"
#include "bnrslide.h"
#include "bnrhardpin.h"
//Analog Slot
Class CAnIOSlot
{
	 void (*CCAnIOSlot)(This);
	 void (*DCAnIOSlot)(This);
Public
     Virtual void (*InitSlot)(This,SHARDSLOT *pSlot);
     Virtual CPin* (*GetPin)(This,BYTE byNumber);
	 void (*Connect)(This,CAnalogPin *pPin);
Private
     CAnalogPin m_pPin[2];
     DECLARE_IMPLEMENT_BASE(CSlot)
}
DECLARE_DEFINITION(CAnIOSlot)
//Analog Slot 4
Class CAnIOSlot4
{
	 void (*CCAnIOSlot4)(This);
	 void (*DCAnIOSlot4)(This);
Public
     Virtual void (*InitSlot)(This,SHARDSLOT *pSlot);
     Virtual CPin* (*GetPin)(This,BYTE byNumber);
	 void (*Connect)(This,CAnalogPin *pPin);
Private
     CAnalogPin m_pPin[DEV_MAX_AI_X20AI4622_PIN];
     DECLARE_IMPLEMENT_BASE(CSlot)
}
DECLARE_DEFINITION(CAnIOSlot4)
//Digital Slot
Class CDgIOSlot
{
	 void (*CCDgIOSlot)(This);
	 void (*DCDgIOSlot)(This);
Public
     Virtual void (*InitSlot)(This,SHARDSLOT *pSlot);
     Virtual CPin* (*GetPin)(This,BYTE byNumber);
     void (*Connect)(This,CDigitalPin *pPin);
Private
     #if MYSYSTEM_ID != 5
	 CDigitalPin m_pPin[32];
     #else
	 CDigitalPin m_pPin[12];
     #endif
	 DECLARE_IMPLEMENT_BASE(CSlot)
}
DECLARE_DEFINITION(CDgIOSlot)
//Counter Slot
Class CCountSlot
{
	 void (*CCCountSlot)(This);
	 void (*DCCountSlot)(This);
Public
	 Virtual void (*InitSlot)(This,SHARDSLOT *pSlot);
	 Virtual CPin* (*GetPin)(This,BYTE byNumber);
	 void (*Connect)(This,CDCounterPin *pPin);
Private
	 CDCounterPin m_pPin[2];
	 DECLARE_IMPLEMENT_BASE(CSlot)
}
DECLARE_DEFINITION(CCountSlot)
//Temperature Slot
Class CTemperatureSlot
{
	void (*CCTemperatureSlot)(This);
	void (*DCTemperatureSlot)(This);
Public
	Virtual void (*InitSlot)(This,SHARDSLOT *pSlot);
	Virtual CPin* (*GetPin)(This,BYTE byNumber);
	void (*Connect)(This,CTemperaturePin *pPin);
Private
	CTemperaturePin m_pPin[2];
	DECLARE_IMPLEMENT_BASE(CSlot)
}
DECLARE_DEFINITION(CTemperatureSlot)
#endif
```

#### bnrauto.h
```c
/********************************************************************
 * COPYRIGHT -- Kontora
 ********************************************************************
 * Program: bnrmain
 * File: bnraninput.h
 * Author: Abramenya
 * Created: January 19, 2009
 *******************************************************************/
#if !defined(__PRI2AUT_H__)
#define __PRI2AUT_H__
#include "typedefs.h"
Class CAuto
{
Public
    void (*CCAuto)(This);
    void (*DCAuto)(This);
    BOOL (*SetState)(This,TStateCode vNewState);
    TStateCode (*GetStateCode)(This);
    BOOL (*HandleEvent)(This,TEvent vEvent);
Protected
    Virtual BOOL (*HandleTask)(This,TTask* pvTask);
    Virtual TStateList* (*GetStateList)(This);
    TState* (*GetState)(This);
Protected
    BYTE v[20];
    TState*  m_pvState;
    TStateCode m_vState;
    DECLARE_IMPLEMENT
}
DECLARE_DEFINITION(CAuto)
#endif //!defined(__AUTOMAT_H__)
```

#### bnrcomputer.h
```c
/********************************************************************
 * COPYRIGHT -- Kontora
 ********************************************************************
 * Program: bnrmain
 * File: bnraninput.h
 * Author: Abramenya
 * Created: January 19, 2009
 *******************************************************************/

#ifndef __COMPUTER_H__
#define __COMPUTER_H__
#include "typedefs.h"
#include "bnrslide.h"
#include "bnraninput.h"
#include "bnrmessage.h"
//#include "bnrtcpdriver.h"
#include "bnrprocmanager.h"
Class CComputer
{
	 void (*CCComputer)(This);
	 void (*DCComputer)(This);
Public
     void   (*Init)(This,SHARDCOMPUTERTABLE *pTable);
     void   (*InitDevModule)(This,SHARDCOMPUTERTABLE *pTable);
	 CSlot* (*CreateSlot)(This,SHARDSLOT *psvSlot);
	 void   (*Connect)(This,CSlot *psSlot);
	 CSlot* (*GetSlot)(This,BYTE byNumber);
	 CSlot* (*CreateSlotCPU_260)(This,SHARDSLOT *psvSlot);
	 CSlot* (*CreateSlotIF_681)(This,SHARDSLOT *psvSlot);
	 CSlot* (*CreateSlot3DI477_6)(This,SHARDSLOT *psvSlot);
	 CSlot* (*CreateSlot3DO477_6)(This,SHARDSLOT *psvSlot);
	 CSlot* (*CreateSlot3AI375_6)(This,SHARDSLOT *psvSlot);
	 CSlot* (*CreateSlotAT2222)(This,SHARDSLOT *psvSlot);
	 CSlot* (*CreateSlotDI2377)(This,SHARDSLOT *psvSlot);
	 CSlot* (*CreateSlot3AI4622)(This,SHARDSLOT *psvSlot);
	 CSlot* (*CreateSlot3AO775_6)(This,SHARDSLOT *psvSlot);
Private
     CSlot **m_pvSlot;
	 BYTE  m_byArmAmout;
     BYTE  m_byComputerType;
     SINT  m_chComputerName[DEV_MAX_TEXT_NAME];
     SINT  m_chProgrammVersion[DEV_MAX_TEXT_NAME];
     SINT  m_chDateOfWrite[DEV_MAX_TEXT_NAME];
	 BYTE  m_bySlotAmout;
     SHARDCOMPUTERTABLE *m_pConfigTable;
	 DECLARE_IMPLEMENT
}
DECLARE_DEFINITION(CComputer)
#endif
```

#### bnrcomserver.h
```c
/********************************************************************
 * COPYRIGHT -- Kontora
 ********************************************************************
 * Program: bnrmain
 * File: bnraninput.h
 * Author: Abramenya
 * Created: January 19, 2009
 *******************************************************************/

#ifndef __COMSERVER_H__
#define __COMSERVER_H__
#include "typedefs.h"
#include "bnrmessage.h"
#include "bnrdebug.h"
#include "bnrcyclicsystem.h"

#ifndef WIN32
//#include <DVFrame.h>
#endif
#ifdef WIN32
void FRM_xopen(FRM_xopen_typ*);
void FRM_close(FRM_close_typ*);
void FRM_gbuf(FRM_gbuf_typ*);
void FRM_rbuf(FRM_rbuf_typ*);
void FRM_robuf(FRM_robuf_typ*);
void FRM_write(FRM_write_typ*);
void FRM_read(FRM_read_typ*);
#endif
#define BUFF_SZ 0x3ff
Class CComServer
{
	 void (*CCComServer)(This);
	 void (*DCComServer)(This);
Public
     //Connection Disconnection Procedure
     void (*Init)(This,SARMINTERFACE *pArm);
Private
	 void (*Close)(This);
     void (*InitSRV)(This);
	 void (*Enable)(This);
	 void (*Disable)(This);
	 BOOL (*Open)(This);
     BOOL (*SendMessage)(This,SMESSAGE *pMsg);
	 BOOL (*GetMessage)(This,SMESSAGE *pMsg);
	 void (*ReceiveThread)(This);
	 void (*SendThread)(This);
	 void (*SynBuff)(This);
	 BOOL (*MakeMsgData)(This,SMESSAGE *pMsg);
	 BOOL (*MakeTextMessage)(This);
	 void (*ATHandler)(This,USINT *pComm,WORD wLen);
	 BOOL (*CopyMessage)(This,WORD wLen,SMESSAGE *pMsg);
	 BYTE (*CreateCRC)(This,BYTE *pMsg,BYTE byLen);
	 INT (*FindText)(This,SINT *pSrc,SINT *pChar);
	 WORD (*CalckSumm)(This,BYTE *pCH,WORD wLen);
	 void (*SendSMessage)(This,BYTE byBox,BYTE byFor,BYTE byType);
	 BOOL (*Connect)(This);
	 BOOL (*Disconnect)(This);
	 void (*SetPortSett)(This);
	 void (*TestMsg)(This);
     Virtual BOOL (*EventHandler)(This,SMESSAGE *pMsg);
     Virtual void (*CyclicProc)(This);
Private
     /*
	 FRM_xopen_typ m_sXOpen;
     XOPENCONFIG m_sConfig;
     FRM_gbuf_typ m_sFrameBuff;
     FRM_rbuf_typ m_sRBuff;
     FRM_write_typ m_sSend;
	 FRM_read_typ m_sRecc;
	 FRM_close_typ m_sClose;
	 FRM_robuf_typ m_sRobuff;
	 */
	 SINT m_chStringDevice[50];
     SINT m_chStringMode[50];
	 SINT m_chStringNewMode[50];
     UINT m_StatusOpen;
	 UINT m_StatusClose;
	 UINT m_StatusWrite;
	 UINT m_StatusRead;
	 UINT m_StatusGetBuffer;
	 UINT m_StatusReleaseBuffer;
	 UINT m_StatusReleaseOutputBuffer;
	 UINT m_SendBufferLength;
	 UINT m_ReadBufferLength;
	 UINT m_Error;

	 USINT m_SendBuffer[300];
	 USINT m_ReadBuffer[300];
	 USINT pb_mBoxDoTextRead[120];
	 //USINT *m_SendBuffer;
	 //USINT *m_ReadBuffer;

	 //BYTE pb_mBoxDoRead[5000];
	 //BYTE pb_mBoxRead[3000];
	 BYTE pb_mBoxCont[BUFF_SZ];
	 WORD w_mBoxSize;
	 WORD w_mBoxCSize;
	 WORD w_mBoxWrite;
	 WORD w_mBoxRead;
	 WORD m_sSize;
     WORD w_lLength;
	 WORD w_lMsgLen;
	 WORD InByteCount_DATA;

	 WORD nWsCount;

	 BYTE m_byType;
	 BYTE m_byRate;
	 BOOL m_blMsgFind;
     STCPADDR m_stTcpAddr;
	 BYTE m_bSrvState;
	 BYTE m_bCliState;
	 SMESSAGE m_sMsg;
	 CMTimer m_nConnTMR;
	 SARMINTERFACE *m_pArm;
	 DECLARE_IMPLEMENT_BASE(CCyclicSystem)
}
DECLARE_DEFINITION(CComServer)
#endif
```

#### bnrconst.h
```c
/********************************************************************
 * COPYRIGHT -- Kontora
 ********************************************************************
 * Program: bnrmain
 * File: bnrconst.h
 * Author: Abramenya
 * Created: January 19, 2009
 *******************************************************************/
#ifndef WIN32
#include <AsDefault.h>
#endif
#ifndef __CONST_H__
#define __CONST_H__
//#define IF_MODEM     0
#define MYSYSTEM_ID  5
#ifdef WIN32
//#define MY_MODEL     0
#endif
//User Define
#ifndef NULL
 #define  NULL 0
#endif
#ifndef WIN32
#define TRUE 1
#define FALSE 0
#endif
//Define System QW
#define ACP_MIN                      6552
#define ACP_MAX                      32760
#define SYSTEM_QTIME                 50
//Event System

#define _DLESS_SHIFT                 0
#define _KPMOD_SHIFT                 0
#define _MSINP_SHIFT                 32
#define _ADMIN_SHIFT                 64
#define _SYSTM_SHIFT                 96
#define _OBSRV_SHIFT                 128
#define _ARMMD_SHIFT                 160
#define _DEBMS_SHIFT                 192
#define _DIRMD_SHIFT                 224
#define _SMSNS_SHIFT                 240

//Data Linc Message
#define EV_DLESS_ARM_RR_REQ	         _DLESS_SHIFT + 0 //Запрос подтверждения к устройству	00
#define EV_DLESS_ARM_RR_IND          _DLESS_SHIFT + 1 //Ответ от устройства на запрос подтверждения	01
#define EV_DLESS_BNR_RR_REQ	         _DLESS_SHIFT + 2 //Запрос подтверждения к АРМ	02
#define EV_DLESS_BNR_RR_IND	         _DLESS_SHIFT + 3 //Ответ от  АРМ на запрос подтверждения	03
#define EV_DLESS_TMRPUT_ARMIN        _DLESS_SHIFT + 4 //Таймер запросов подтверждений	04
#define EV_DLESS_TMRGET_ARMIN        _DLESS_SHIFT + 5 //Таймер на ответ на запрос подтверждения к устройству	05

#define EV_MCSET_IN00                _MSINP_SHIFT + 0
#define EV_MCSET_IN01                _MSINP_SHIFT + 1
#define EV_MCSET_IN02                _MSINP_SHIFT + 2
#define EV_MCSET_IN03                _MSINP_SHIFT + 3
#define EV_MCSET_IN04                _MSINP_SHIFT + 4
#define EV_MCSET_IN05                _MSINP_SHIFT + 5
#define EV_MCSET_IN06                _MSINP_SHIFT + 6
#define EV_MCSET_IN07                _MSINP_SHIFT + 7
#define EV_MCSET_IN08                _MSINP_SHIFT + 8
#define EV_MCSET_IN09                _MSINP_SHIFT + 9
#define EV_MCSET_IN10                _MSINP_SHIFT + 10
#define EV_MCSET_IN11                _MSINP_SHIFT + 11
#define EV_MCSET_IN12                _MSINP_SHIFT + 12
#define EV_MCSET_IN13                _MSINP_SHIFT + 13
#define EV_MCSET_IN14                _MSINP_SHIFT + 14
#define EV_MCSET_IN15                _MSINP_SHIFT + 15
#define EV_MCSET_IN16                _MSINP_SHIFT + 16
#define EV_MCSET_IN17                _MSINP_SHIFT + 17
#define EV_MCSET_IN18                _MSINP_SHIFT + 18
#define EV_MCSET_IN19                _MSINP_SHIFT + 19
#define EV_MCSET_IN20                _MSINP_SHIFT + 20
#define EV_MCSET_IN21                _MSINP_SHIFT + 21
#define EV_MCSET_IN22                _MSINP_SHIFT + 22
#define EV_MCSET_IN23                _MSINP_SHIFT + 23
#define EV_MCSET_IN24                _MSINP_SHIFT + 24
#define EV_MCSET_IN25                _MSINP_SHIFT + 25
#define EV_MCSET_IN26                _MSINP_SHIFT + 26
#define EV_MCSET_IN27                _MSINP_SHIFT + 27
#define EV_MCSET_IN28                _MSINP_SHIFT + 28
#define EV_MCSET_IN29                _MSINP_SHIFT + 29
#define EV_MCSET_IN30                _MSINP_SHIFT + 30
#define EV_MCSET_IN31                _MSINP_SHIFT + 31

//Admin Message
#define EV_ADMIN_ARM_CONFIG_REQ	     _ADMIN_SHIFT + 0 //Передать таблицу конфигурации для драйвера АРМ	64
#define EV_ADMIN_SYS_CONFIG_REQ	     _ADMIN_SHIFT + 1 //Передать таблицу конфигурации для драйвера системы	65
#define EV_ADMIN_SYS_CONFIG_IND	     _ADMIN_SHIFT + 2 //Запросить таблицу конфигурации для системы сенсоров
#define EV_ADMIN_SYS_READY_IND	     _ADMIN_SHIFT + 3 //Система готова к работе
#define EV_ADMIN_ARM_CONN_IND	     _ADMIN_SHIFT + 4 //АРМ подключен	66
#define EV_ADMIN_ARM_DISC_IND	     _ADMIN_SHIFT + 5 //АРМ отключен	67

#define EV_ADMIN_SET_ALM_HILEV_REQ   _ADMIN_SHIFT + 6 //Авария превышения верхнего ав. предела 	68
#define EV_ADMIN_REM_ALM_HILEV_REQ	 _ADMIN_SHIFT + 7 //Устранение аварии превышения верхнего ав. предела 	69

#define EV_ADMIN_SET_ALM_LOLEV_REQ	 _ADMIN_SHIFT + 8 //Авария превышения нижнего ав. предела 	70
#define EV_ADMIN_REM_ALM_LOLEV_REQ	 _ADMIN_SHIFT + 9 //Устранение аварии превышения нижнего ав. предела 	71
#define EV_ADMIN_ASK_CONF_TIM_IND	 _ADMIN_SHIFT + 10 //Таймер запроса конфигурации
#define EV_ADMIN_ARM_STOP_REQ	     _ADMIN_SHIFT + 11
#define EV_ADMIN_TMR_SSTATE_IND	     _ADMIN_SHIFT + 12
#define EV_ADMIN_ARM_READY_REQ	     _ADMIN_SHIFT + 13

#define EV_ADMIN_OPER_LO_REQ	     _ADMIN_SHIFT + 14
#define EV_ADMIN_OPER_HI_REQ	     _ADMIN_SHIFT + 15

//System Message
#define EV_SYSTM_CLOSE_INPOTRS_REQ	 _SYSTM_SHIFT + 0 //Закрыть все входные порты 	96
#define EV_SYSTM_OPEN_INPOTRS_REQ	 _SYSTM_SHIFT + 1 //Открыть все входные порты	97
#define EV_SYSTM_CLOSE_OUTPOTRS_REQ	 _SYSTM_SHIFT + 2 //Закрыть все выходные порты	98
#define EV_SYSTM_OPEN_OUTPOTRS_REQ	 _SYSTM_SHIFT + 3 //Открыть все выходные порты	99
#define EV_SYSTM_STOP_JOB_REQ	     _SYSTM_SHIFT + 4 //Остановить задачу	100
#define EV_SYSTM_START_JOB_REQ	     _SYSTM_SHIFT + 5 //Запустить задачу	101
#define EV_SYSTM_FREQ_JOB_REQ	     _SYSTM_SHIFT + 6 //Установить частоту вызова задачи	102
#define EV_SYSTM_INIT_OBS_REQ	     _SYSTM_SHIFT + 7 //Проинициализировать модуль наблюдения
#define EV_SYSTM_INIT_OBS_IND	     _SYSTM_SHIFT + 8 //Ответ на команду инициализации
#define EV_SYSTM_RESET_BOARD_IND	 _SYSTM_SHIFT + 9 //Запрос на сброс
#define EV_SYSTM_RESET_TIM_BRD_IND	 _SYSTM_SHIFT + 10 //Сброс по таймеру

//Observe System Message
#define EV_OBSRV_GET_INOUT_SDATA_IND _OBSRV_SHIFT + 0 //Вернуть входное и выходное значение сенсоров	148
#define EV_OBSRV_GET_OUT_DATA_IND    _OBSRV_SHIFT + 1
#define EV_OBSRV_START_DATA_PROC_REQ _OBSRV_SHIFT + 2 //Инициировать процесс передачиданных с частотой X
#define EV_OBSRV_STOP_DATA_PROC_REQ  _OBSRV_SHIFT + 3 //Остановить процесс передачиданных с частотой X
#define EV_OBSRV_REFR_TIM_PROC_IND   _OBSRV_SHIFT + 4 //Таймер обновления данных
#define EV_OBSRV_SET_MODE_REQ	     _OBSRV_SHIFT + 5 //Установить режим
#define EV_OBSRV_GET_MODE_REQ    	 _OBSRV_SHIFT + 6 //Запросить режим
#define EV_OBSRV_GET_MODE_IND    	 _OBSRV_SHIFT + 7 //Вернуть режим
#define EV_OBSRV_GET_DMC_DATA_IND    _OBSRV_SHIFT + 8 //Вернуть состояние лог модуля
#define EV_OBSRV_RFLASH_SAVE_REQ     _OBSRV_SHIFT + 9 //Сохранение контекста
#define EV_OBSRV_REMFLS_SAVE_REQ     _OBSRV_SHIFT + 10 //Сохранение контекста в другом процессе

//Arm Module Message
#define EV_MCREM_IN00                _ARMMD_SHIFT + 0
#define EV_MCREM_IN01                _ARMMD_SHIFT + 1
#define EV_MCREM_IN02                _ARMMD_SHIFT + 2
#define EV_MCREM_IN03                _ARMMD_SHIFT + 3
#define EV_MCREM_IN04                _ARMMD_SHIFT + 4
#define EV_MCREM_IN05                _ARMMD_SHIFT + 5
#define EV_MCREM_IN06                _ARMMD_SHIFT + 6
#define EV_MCREM_IN07                _ARMMD_SHIFT + 7
#define EV_MCREM_IN08                _ARMMD_SHIFT + 8
#define EV_MCREM_IN09                _ARMMD_SHIFT + 9
#define EV_MCREM_IN10                _ARMMD_SHIFT + 10
#define EV_MCREM_IN11                _ARMMD_SHIFT + 11
#define EV_MCREM_IN12                _ARMMD_SHIFT + 12
#define EV_MCREM_IN13                _ARMMD_SHIFT + 13
#define EV_MCREM_IN14                _ARMMD_SHIFT + 14
#define EV_MCREM_IN15                _ARMMD_SHIFT + 15
#define EV_MCREM_IN16                _ARMMD_SHIFT + 16
#define EV_MCREM_IN17                _ARMMD_SHIFT + 17
#define EV_MCREM_IN18                _ARMMD_SHIFT + 18
#define EV_MCREM_IN19                _ARMMD_SHIFT + 19
#define EV_MCREM_IN20                _ARMMD_SHIFT + 20
#define EV_MCREM_IN21                _ARMMD_SHIFT + 21
#define EV_MCREM_IN22                _ARMMD_SHIFT + 22
#define EV_MCREM_IN23                _ARMMD_SHIFT + 23
#define EV_MCREM_IN24                _ARMMD_SHIFT + 24
#define EV_MCREM_IN25                _ARMMD_SHIFT + 25
#define EV_MCREM_IN26                _ARMMD_SHIFT + 26
#define EV_MCREM_IN27                _ARMMD_SHIFT + 27
#define EV_MCREM_IN28                _ARMMD_SHIFT + 28
#define EV_MCREM_IN29                _ARMMD_SHIFT + 29
#define EV_MCREM_IN30                _ARMMD_SHIFT + 30
#define EV_MCREM_IN31                _ARMMD_SHIFT + 31

//Debug Message
#define EV_DEBMS_DEBOUT_IND          _DEBMS_SHIFT + 0

//Dir Module
#define EV_DIRMD_CONN_STAT_SNS_IND   _DIRMD_SHIFT + 0 //Установить соединение с сенсором
#define EV_DIRMD_DISC_STAT_SNS_IND   _DIRMD_SHIFT + 1 //Разорвать соединение с сенсором
#define EV_DIRMD_CONN_STAT_START_IND _DIRMD_SHIFT + 2 //Запустить проседуру сбора данных с периодом в секундах
#define EV_DIRMD_CONN_STAT_STOP_IND  _DIRMD_SHIFT + 3 //Остановить проседуру сбора данных
#define EV_DIRMD_REFR_TIM_PROC_IND   _DIRMD_SHIFT + 4 //Таймер сбора статистических данных
#define EV_DIRMD_STAT_DATA_IND       _DIRMD_SHIFT + 5 //Массив статистических данных за период
#define EV_DIRMD_GET_PARAM_REQ       _DIRMD_SHIFT + 6 //Запросить араметры сенсора
#define EV_DIRMD_SET_TANK_REQ        _DIRMD_SHIFT + 7

#define EV_SENSR_GET_SNPARAM_REQ     _SMSNS_SHIFT + 0  //Запросить у датчика параметры
#define EV_SENSR_GET_SNPARAM_IND     _SMSNS_SHIFT + 1  //Вернуть параметры датчика
#define EV_SENSR_SET_SNPARAM_REQ     _SMSNS_SHIFT + 2  //Установить параметры датчика
#define EV_SENSR_SET_PDPARAM_REQ     _SMSNS_SHIFT + 3  //Установить параметры ПИД
#define EV_SENSR_GET_PDPARAM_IND     _SMSNS_SHIFT + 4  //Вернуть параметры ПИД
#define EV_SENSR_SET_DIGT_OUT_REQ    _SMSNS_SHIFT + 5  //Подать значение на выход
#define EV_SENSR_SET_DIGT_PULCE_REQ  _SMSNS_SHIFT + 6  //Подать импульс

#define EV_SENSR_TMR_SAHI            _SMSNS_SHIFT + 5
#define EV_SENSR_TMR_RAHI            _SMSNS_SHIFT + 6
#define EV_SENSR_TMR_SALO            _SMSNS_SHIFT + 7
#define EV_SENSR_TMR_RALO            _SMSNS_SHIFT + 8

/////////////////////////////////////////////////////////////////////////////
//BEGIN:                      Level Module 101                             //
/////////////////////////////////////////////////////////////////////////////
#define PL_DATA_IND                  _KPMOD_SHIFT + 17
#define PL_DATA_REQ                  _KPMOD_SHIFT + 18
//Primitives For Data Linc Level
#define DL_DATA_IND                  _KPMOD_SHIFT + 19
#define DL_DATA_REQ                  _KPMOD_SHIFT + 20
#define DL_DATA_RES                  _KPMOD_SHIFT + 21
//Primitives For Data Physic Level
#define PH_DATA_IND                  _KPMOD_SHIFT + 22
#define PH_DATA_REQ                  _KPMOD_SHIFT + 23

#define PH_CONN_REQ                  _KPMOD_SHIFT + 24
#define PH_DISC0_REQ                 _KPMOD_SHIFT + 25
#define PH_DISC_REQ                  _KPMOD_SHIFT + 26
#define PH_CONN_IND                  _KPMOD_SHIFT + 27
#define PH_DISC_IND                  _KPMOD_SHIFT + 28

#define PH_DATA_RES                  _KPMOD_SHIFT + 29
#define PH_DATA1_RES                 _KPMOD_SHIFT + 30

#define PH_DATA_CON                  _KPMOD_SHIFT + 31
#define PH_DATA_NCON                 _KPMOD_SHIFT + 32
#define PH_DATA_REP                  _KPMOD_SHIFT + 33
#define PH_DATA_RD_CON               _KPMOD_SHIFT + 34

#define PH_DATA_UP_REQ               _KPMOD_SHIFT + 35
#define PH_INIT_REQ                  _KPMOD_SHIFT + 36
#define PH_CALL_REQ                  _KPMOD_SHIFT + 37
#define PH_TIME_ST_REQ               _KPMOD_SHIFT + 38
#define PH_CLOSE_PORT_REQ            _KPMOD_SHIFT + 39
#define PH_INIT_PORT_REQ             _KPMOD_SHIFT + 40
#define PH_SETT_KPID_REQ             _KPMOD_SHIFT + 41
#define PH_VS0_REQ                   _KPMOD_SHIFT + 42
#define PH_VS1_REQ                   _KPMOD_SHIFT + 43
#define PH_SCMD_REQ                  _KPMOD_SHIFT + 44

#define PH_DATA_RD_REQ               _KPMOD_SHIFT + 65
#define PH_DATA_WR_REQ               _KPMOD_SHIFT + 66
#define EV_TMR_SRR_REQ               _KPMOD_SHIFT + 67 //Таймер SRR
#define EV_TMR_SSC_REQ               _KPMOD_SHIFT + 68 //Таймер SSC
#define EV_TMR_DISC_REQ              _KPMOD_SHIFT + 69 //Таймер DISC
#define EV_TMR_CNRP_REQ              _KPMOD_SHIFT + 70 //Таймер DISC
#define EV_TMR_PUCM_REQ              _KPMOD_SHIFT + 71 //Таймер DISC
#define EV_TMR_SDIS_REQ              _KPMOD_SHIFT + 72 //Таймер DISC
#define EV_TMR_RCAL_REQ              _KPMOD_SHIFT + 73 //Таймер DISC
#define EV_TMR_OUT_REQ               _KPMOD_SHIFT + 74 //Таймер DISC
#define EV_CHNG_PIN_REQ              _KPMOD_SHIFT + 75 //Таймер DISC
//Сообщения пролива
#define EV_START_WSY_REQ             _KPMOD_SHIFT + 76 //Запуск модуля
#define EV_HAND_STOP_WSY_REQ         _KPMOD_SHIFT + 77 //Ручной останов
#define EV_HAND_START_WSY_REQ        _KPMOD_SHIFT + 78 //Ручной старт
#define EV_TMR_WTOP_REQ              _KPMOD_SHIFT + 79 //Таймер Ожидания Операционного режима
#define EV_TMR_OPER_REQ              _KPMOD_SHIFT + 80 //Таймер Операционного режима
#define EV_TMR_WTST_REQ              _KPMOD_SHIFT + 81 //Таймер Ожидания Успокоения Жидкости
#define EV_CT_OFF_REQ                _KPMOD_SHIFT + 82 //Счет завершен

#define PL_ASDU_DC0_IND              46
#define PL_ASDU_NVA_IND              48

//Events From PH Level
#define EV_RESET_SC00_IND            _KPMOD_SHIFT + 0  //Перезапуск удаленной связи
#define EV_DATA_SC03_IND             _KPMOD_SHIFT + 3  //Данные пользователя с повтором
#define EV_DATAN_SC04_IND            _KPMOD_SHIFT + 4  //Данные пользователя без повтора
#define EV_STJOIN_RR09_IND           _KPMOD_SHIFT + 9  //Запрос статуса связи
#define EV_DATA1_RR10_IND            _KPMOD_SHIFT + 10 //Запрос данных пользователя класса 1
#define EV_DATA2_RR11_IND            _KPMOD_SHIFT + 11 //Запрос данных пользователя класса 2
//Events For PH Level
#define EV_ACK_SC00_CON              _KPMOD_SHIFT + 0  //ACK: положительное подтверждение
#define EV_NACK_SC01_CON             _KPMOD_SHIFT + 1  //NACK: сообщение не принято, линия занята
#define EV_ACK_RR08_RES              _KPMOD_SHIFT + 8  //Данные пользователя
#define EV_NACK_RR08_RES             _KPMOD_SHIFT + 9  //NACK: затребованные данные недоступны
#define EV_STJOIN_RR08_RES           _KPMOD_SHIFT + 11 //Статус связи или требование доступа

//State For KP Machine
#define MKP_NULL_ST00                0
#define MKP_CONN_ST01                1
#define MKP_DISC_ST02                2

//State For 101 Machine
#define M101_NULL_ST00               0
#define M101_CONN_ST01               1
#define M101_DISC_ST02               2

//State For GSM Machine
#define MGSM_DISC_ST00               0
#define MGSM_CONN_ST01               1
#define MGSM_WCON_ST02               2

#define MSG_LONG_CODE 0x68
#define MSG_SHRT_CODE 0x10

#define MSG_ASDU_DQ_CODE 46
#define MSG_ASDU_WR_CODE 48
#define MSG_ASDU_RD_CODE 102
#define MSG_TIME_ST_CODE 103

#define MSK_RES 0x80
#define MSK_PRM 0x40
#define MSK_FCB 0x20
#define MSK_FCV 0x10

/////////////////////////////////////////////////////////////////////////////
//END;                        Level Module 101                             //
/////////////////////////////////////////////////////////////////////////////

//Para Pid Init
#define SNS_PARA_INI 0
#define SNS_PIDC_INI 1
#define SNS_SENS_INI 2
#define SNS_SENS_CTR 3
#define SNS_SENS_OUT 4
//Para Init
#define PR_Y_max    0
#define PR_Y_min    1
#define PR_dY_max   2
#define PR_Kp       3
#define PR_Tn       4
#define PR_Tv       5
#define PR_Tf       6
#define PR_Kw       7
#define PR_Kfbk     8
#define PR_PrEn     9
//Pid Init
#define PR_W        10
#define PR_X        11
#define PR_A        12
#define PR_Y_man    13
#define PR_out_mode 14
#define PR_PidEn    15
//Sensor Init
#define PR_LO       16
#define PR_HI       17
#define PR_ALO      18
#define PR_AHI      19
#define PR_PLO      20
#define PR_PHI      21
#define PR_ACO      22
#define PR_PDO      23
#define PR_RST      24
#define PR_INI      25
#define PR_INC_IN   26
#define PR_DEC_IN   27
#define PR_Out_En   28
#define PR_Inp_En   29
#define PR_Lay_En   30
#define PR_OPN_GT   31
#define PR_OMIN     32
#define PR_OMAX     33
#define PR_PMODE    34
#define PR_OMODE    35
#define PR_STOP_GT  36
#define PR_ACM      37
#define PR_OTIME    38
#define PR_EnFlt    39
#define PR_PRC_GT   40

#define EV_SMSNS_SET_PARAM_REQ       _SMSNS_SHIFT + 0 //Установить параметры   //Len Type LenParam Param

//Timer Message
#define EV_TMR000_ADMIN     26
#define EV_TMRTIN_SYSTM     27
#define EV_TMRTIN_ARMIN     28

//Debug Flags
#define DEB_OUT_CYC_ADMIN 0x01
#define DEB_OUT_CYC_SYSTM 0x02
#define DEB_OUT_CYC_OBSRV 0x04
#define DEB_OUT_PMAN_STAT 0x08
#define DEB_OUT_OBSR_COMM 0x10
#define DEB_OUT_DIRC_COMM 0x20

#define DEB_OUT_BOX_ADMIN 0x40
#define DEB_OUT_BOX_SYSTM 0x80
#define DEB_OUT_BOX_OBSRV 0x100

//Timer Constant
enum _enTimeConst
{
	    /*
		T05SEC =  5*100/SYSTEM_QTIME,
	    T1SEC  = 10*100/SYSTEM_QTIME,
		T2SEC  = 20*100/SYSTEM_QTIME,
		T3SEC  = 30*100/SYSTEM_QTIME,
        T4SEC  = 40*100/SYSTEM_QTIME,
		T5SEC  = 50*100/SYSTEM_QTIME,
		T6SEC  = 60*100/SYSTEM_QTIME,
        T7SEC  = 70*100/SYSTEM_QTIME,
		T8SEC  = 80*100/SYSTEM_QTIME,
        T9SEC  = 90*100/SYSTEM_QTIME,
		T10SEC =100*100/SYSTEM_QTIME,
		*/
  	    T05SEC =  5,
		T1SEC  = 10,
		T2SEC  = 20,
		T3SEC  = 30,
        T4SEC  = 40,
		T5SEC  = 50,
		T6SEC  = 60,
        T7SEC  = 70,
		T8SEC  = 80,
        T9SEC  = 90,
		T10SEC =100,
};

//Max Switching In Direction
#if MYSYSTEM_ID !=5
#define DEV_AMT_SWC_IDIR      20
#else
#define DEV_AMT_SWC_IDIR      150
#endif

//Max Out Gate
#define DEV_AMT_GATE_SNS      5
//Max Base Gate
#define BASE_GTE              6683
#define MAX_GTE               5100
//Max Out Gate TYPE
enum _tagTypeGate
{
	IDLES_GTE=0,
	SMART_GTE,
};
enum _tagTeleSignal
{
	TS=0,
	TI,
	TU,
	TIS,
	TC,
	TPR,
	TTM,
	TF,
	TKP,
	TPU,
	TVS,
	TLV,
	TPL,
	TMR,
	TAL,
	TOS,
};
//Max Direction In System
#define DEV_AMT_DIR_INST      1
//Proc Manager State
enum _enManagerState
{
        DEV_PROC_STT_ONN = 0,
        DEV_PROC_STT_OFF,
};
//System Queue ID
#define DEV_ARMIN_BOX_ID      0
#define DEV_ARMOT_BOX_ID      1
#define DEV_ARMAD_BOX_ID      2
#define DEV_SYSTM_BOX_ID      3
#define DEV_ADMIN_BOX_ID      4
#define DEV_KPMDL_BOX_ID      5
#define DEV_101MD_BOX_ID      6
#define DEV_GSMMD_BOX_ID      7
#define DEV_RSMMD_BOX_ID      8
#define DEV_RSBUF_BOX_ID      9
#define BOX_L4                10
#define BOX_REG               11
#define BOX_L4_1              12

#define DEV_RSVBS0_BOX_ID     13
#define DEV_RSVS0MMD_BOX_ID   14

#define DEV_RSVBS1_BOX_ID     15
#define DEV_RSVS1MMD_BOX_ID   16

#define DEV_TCPRM_BOX_ID      17
#define DEV_TCPBF_BOX_ID      18
#define DEV_MSMDL_BOX_ID      19

//System Queue Size
#define DEV_SYSTM_BOX_SZ      512    // No
#define DEV_ADMIN_BOX_SZ      512    // No
#define DEV_ARMIN_BOX_SZ      512    // No
#define DEV_ARMOT_BOX_SZ      512    // Yes
#define DEV_ARMAD_BOX_SZ      1*512  // No
#define DEV_KPMDL_BOX_SZ      2*512  // Yes
#define DEV_101MD_BOX_SZ      2*512  // Yes
#define DEV_RSMMD_BOX_SZ      4*1024  // Yes
#define DEV_RSBUF_BOX_SZ      4*1024  // Yes
#define BOX_L4_SZ             10*1024 // Yes
#define BOX_REG_SZ            2*512  // Yes
#define BOX_L4_1_SZ           3*1024 // Yes

//Max Message Size
#define DEV_MAX_MSG_SIZE      256
//Max Cyclic Proc
#define DEV_MAX_CYC_PROC      10
//Max System Timers
#define DEV_MAX_SYS_TIMR      30
//State Of Thread
#define DEV_CJOB_ST_SUSP      0
#define DEV_CJOB_ST_RESM      1
#define DEV_JOB_MAX_PROD      10
#define DEV_JOB_MAX_PNME      50
//Max TCP Port
#define DEV_MAX_TCP_PORT      5
#define DEV_MAX_ARM_PORT      5
//Driver State
#define DRV_ST_DISC           0x00
#define DRV_ST_CONN           0x01
#define DRV_ST_NULL           0x02
#define DRV_ST_OPEN           0x03
//Port Type
enum _enType
{
   	    DEV_ARM_PORT_TCP=0,
        DEV_ARM_PORT_UDP,
        DEV_ARM_PORT_COM232,
        DEV_ARM_PORT_COM458,
        DEV_ARM_PORT_USB,
        DEV_SYS_INTERFACE,
};
//Port Rate
enum _enRate
{
        DEV_ARM_RATE_9600=0,
        DEV_ARM_RATE_14400,
        DEV_ARM_RATE_38400,
        DEV_ARM_RATE_57600,
        DEV_ARM_RATE_115200,
        DEV_ARM_RATE_10MBS,
        DEV_ARM_RATE_100MB,
};
//Computer Type
#define DEV_CPU_TYPE_PS260    0
#define DEV_CPU_TYPE_X20      0
#define DEV_MAX_TEXT_NAME     50
//Maximum amount slot in device
#define DEV_MAX_SLOTS_PS260   20
#define DEV_CUR_SLOTS_PS260   4
#define DEV_MAX_DEFAULT_PIN   32
//Max Pin In Device
#define DEV_MAX_AI_3AI375_PIN 8
#define DEV_MAX_AO_3AO775_PIN 8
#define DEV_MAX_DI_3DI477_PIN 32
#define DEV_MAX_DO_3DO760_PIN 8
//Max Pin In Device
#define DEV_MAX_DI_X20DM9371_PIN 12
#define DEV_MAX_DI_X20DI9371_PIN 12
#define DEV_MAX_DI_X20DI2377_PIN 2
#define DEV_MAX_DO_X20DM9322_PIN 12
#define DEV_MAX_DO_X20DO9322_PIN 12
#define DEV_MAX_DO_X20DO9321_PIN 12
#define DEV_MAX_AI_X20AI4622_PIN 4
#define DEV_MAX_AI_X20AI2622_PIN 2
#define DEV_MAX_AO_X20AO4622_PIN 4
#define DEV_MAX_AT_X20AT2222_PIN 2
#define DEV_MAX_DI_X20DI2377_PIN 2
//Type Of Device
enum _tagDeviceType
{
        DEV_DEFAULT_PORT=0,
        DEV_PLC_CPU_260,
		DEV_PLC_CPU_X20,
		DEV_TCPCOM_IF_681,
		DEV_PWCOM_PS9500,
		DEV_COM_CS1020,
		DEV_AI_3AI375_6,
		DEV_AI_X20AI4622,
		DEV_AI_X20AI2622,
		DEV_AO_3AO775_6,
		DEV_AO_X20AO4622,
		DEV_DI_3DI477_6,
		DEV_DI_X20DM9371,
		DEV_DI_X20DI9371,
		DEV_DI_X20DI2377,
		DEV_DO_3DO760_6,
		DEV_DO_X20DM9322,
		DEV_DO_X20DO9321,
		DEV_AT_X20AT2222
};
//Hard Pin State
enum _tagPinState
{
		PIN_STATE_DEF=0,
		PIN_STATE_ONN,
		PIN_STATE_OFF,
		PIN_STATE_TRI,
};
//Out State
enum _tagInOutState
{
	    ST_INIT =0,
		ST_OPEN =1,
		ST_CLOS=2,
		ST_NULL =3,
};
//Type Of Hard Pin
enum _tagPinType
{
		PIN_DEFAULT_PIN=0,
		PIN_AN_INOT_INT,
		PIN_DG_INOT_BOL,
		PIN_ST_INPT_USI,
		PIN_ST_OUTP_USI,
};
#define MAX_POINTER 20
#define BNR_MAX_DIRECTION 16
#define BNR_MAX_CHANNELS  32
//Sensor State
#define ST00_SNS_NULL     0x00
#define ST01_SNS_OPEN     0x01
#define ST02_SNS_CLOS     0x02
//Alarm State
#define ALM_ST_ONN        0x00
#define ALM_ST_OFF        0x01

 //Determination of the modules
enum _enDirection
{
		MDL_ADMIN = 0,
		MDL_HCOMM,
		MDL_ARMMD,
		MDL_SYSTM,
		MDL_DIRMD,
		MDL_CHANN,
		MDL_SENSR,
		MDL_PSENS,
		MDL_TSENS,
		MDL_LSENS,
		MDL_SSENS,
		MDL_COMPT,
		MDL_WRDIN,
		MDL_DINPT,
		MDL_DOUTP,
		MDL_ANINP,
		MDL_ANOUT,
		MDL_CMMIN,
		MDL_TCPDR,
		MDL_COMDR,
		MDL_DEBMS,
		MDL_DLESS,
		MDL_OBSRV,
		MDL_TRSIT,
		MDL_ARMSY,
		MDL_TPIDT,
		DIR_KPMOD,
		DIR_101MD,
		DIR_GSMDL,
		DIR_PHMDL,

		DIR_PHTOGSM,
		DIR_PHTOPH,
		DIR_PHTO101,
		DIR_PHTO101P,
		DIR_GSMTO101P,
		DIR_GSMTO101M,
		DIR_101TOGSM,
		DIR_101TOPH,
		DIR_101TOKP,
		DIR_101TO101,
		DIR_KPTO101,
		DIR_KPTOKP,
		DIR_GSMTOPH,
		DIR_PHTOKP,
		DIR_KPTOPH,
		DIR_TCPTOTCP,
		DIR_MSTOTCP,
		DIR_MSTOPH,
		DIR_PHTOMS,
		DIR_MSTOMS,
		DIR_MSTODV,
		DIR_OSYTOOSY,
};
enum _tagSensorOutMode
{
	    NO=0,
        NZ,
};
//Sensor Proc Mode
enum _tagSensorProcMode
{
	    SDIR = 0,
	    SINV,
};
//Sensor Mode
enum _tagSensorMode
{
        SNS_MD_LOOP = 0,
        SNS_MD_AUTO,
        SNS_MD_MANU,
};
//Sensor Type
enum _tagSensorType
{
	    SNS_SMART = 0,
	    SNS_IDLES,
	    SNS_EMPTY,
};
enum _tagParamType
{
	    P_LEVEL=0,
	    P_TEMPR,
        P_PRESS,
};
//SlotNumber
enum _enSlotNumber
{
	    SL00 = 0,
		SL01,
		SL02,
		SL03,
		SL04,
		SL05,
		SL06,
		SL07,
		SL08,
		SL09,
		SL10,
		SL11,
		SL12,
		SL13,
		SL14,
		SL15,
		SLDF,
};
//Pin Number
enum _enPinNumber
{
	    PN00 = 0,
		PN01,
		PN02,
		PN03,
		PN04,
		PN05,
		PN06,
		PN07,
		PN08,
		PN09,
		PN10,
		PN11,
		PN12,
		PN13,
		PN14,
		PN15,
		PN16,
		PN17,
		PN18,
		PN19,
		PN20,
		PN21,
		PN22,
		PN23,
		PN24,
		PN25,
		PN26,
		PN27,
		PN28,
		PN29,
		PN30,
		PN31,
		PNDF,
};
//Soft Switching Command
enum _enSwitchCommand
{
	    SWC_CMD_INP_OUT=0,
        SWC_CMD_INP_INP,
		SWC_CMD_SMR_CON,
		SWC_CMD_IDL_CON,
		SWC_CMD_EMT_CON,
		SWC_CMD_LOG_CON,
};
//Automat
//
enum _enGateId
{
	GT0=0,
	GT1,
	GT2,
};
//Sensor State
#define SNS_STATE_FREE 0
#define SNS_STATE_PROC 1
//Sensor Command
#define TMR_SET_ALM_HI 0
#define TMR_REM_ALM_HI 1
#define TMR_SET_ALM_LO 2
#define TMR_REM_ALM_LO 3
enum _enSensorCommand
{
	CMD_OPENGATE=0,
    CMD_SETSTATE,
	CMD_SEND,
	CMD_SETVALUE,
	CMD_TIMERON,
	CMD_TIMEROFF,
	CMD_MOV,
	CMD_CMP,
	CMD_REPMSG,
	CMD_PUTMSG,
	CMD_INCC,
	CMD_CHKBUF,
	CMD_CHECKTI,
	CMD_CODE,
	CMD_START_FC,
	CMD_STOP_FC,
	CMD_START_PU,
	CMD_STOP_PU,
	CMD_START_CT,
	CMD_STOP_CT,
};
//Sensor Value
enum _tagAutoValue
{
	INC_INP=0,
	STATE,
};
enum _enCompareValue
{
 	JE=0,
	JNE,
	JA,
	JBE,
};
//Reg Keys
enum _enRegParamAddres
{
	REG_KPPAR_ADDR=0,
    REG_PORTT_ADDR,
    REG_HARDT_ADDR,
    REG_SOFTI_ADDR,
    REG_SOFTS_ADDR,
    REG_SOFTU_ADDR,
    REG_SOFTR_ADDR,
};
enum _enKpCommand
{
	CKP_SETT_KPID=4,
	CKP_SETT_TIME=9,
	CKP_CLSE_PORT,
	CKP_SAVE_SETT,
	CKP_REST_BORD,
	CKP_REST_12BR,
	CKP_STOP_REST,
	CKP_FREE_BXL4,
	CKP_SETT_BL41,
	CKP_AUTO_PSWR,
	CKP_REMT_DISC,
	CKP_SVAL_PINS,
	CKP_SVAL_SLOT,
	CKP_STRT_CHTM,
	CKP_STOP_CHTM,
	CKP_INIT_PORT,
};
//Store Buffers Mode
enum _enStoreMode
{
	SBM_TIUNLOAD = 0x01,
	SBM_TSUNLOAD = 0x02,
	SBM_TUUNLOAD = 0x04,
	SBM_TRUNLOAD = 0x08,
};
//Store Buffers Mode
enum _enTParity
{
	NOPAR=0,
	EVEN,
	ODD,
};
enum _enTData
{
	D_7=0,
	D_8,
};
enum _enTStop
{
	S_1=0,
	S_1_5,
	S_2,
};
enum _enTSPtiority
{
	PRI_LO=0,
	PRI_HI,
};
enum _enTeleObjectState
{
	EN_CLOSE=0,
	EN_OPEN,
	EN_LOCK,
	EN_UNLOCK,
};
enum _enTSAlarmMode
{
	EN_LO_TO_HI=0,
	EN_HI_TO_LO,
	EN_AL_TO_AL,
};
enum _enTUType
{
	EN_INVERT=0,
	EN_DIRECT,
};
#endif
```

#### bnrcyclicsystem.h
```c
/********************************************************************
 * COPYRIGHT -- Kontora
 ********************************************************************
 * Program: bnrmain
 * File: bnraninput.h
 * Author: Abramenya
 * Created: January 19, 2009
 *******************************************************************/

#ifndef __CYCLICSYSTEM_H__
#define __CYCLICSYSTEM_H__
#include "typedefs.h"
#include "bnrmessage.h"
#include "bnrpob.h"
//#include "bnrauto.h"
#include "bnrmytimer.h"
Class CCyclicSystem
{
	 void (*CCCyclicSystem)(This);
	 void (*DCCyclicSystem)(This);
Public
     void (*Create)(This,SINT* chProcName,BYTE byStateProc,BYTE byPeriod);
     void (*CreateSuspend)(This,SINT* chProcName,BYTE byPeriod);
     void (*Start)(This);
	 void (*Stop)(This);
	 void (*SetStateProc)(This,BYTE byStateProc);
	 void (*SetBoxID)(This,BYTE byID);
	 void (*SetPeriod)(This,BYTE byPeriod);
	 void (*SetName)(This,SINT* chProcName);
	 void (*SendMessageData)(This,BYTE byBox,BYTE byFor,BYTE byType,PVOID pData,WORD wLen);
	 void (*SendMessageData1)(This,BYTE byBox,BYTE byFor,BYTE byType,SMESSAGE *pInMsg, PVOID pData,WORD wLen);
	 BYTE (*GetStateProc)(This);
	 WORD (*GetWordParam)(This,BYTE *pbyParam,BYTE *pbyOut);
     Virtual void (*CyclicProc)(This);
	 Virtual BOOL (*GetMessage)(This);
	 Virtual BOOL (*EventHandler)(This,SMESSAGE *pMsg);

	 void (*SetMsgAuto)(This,SMESSAGE*);
	 BOOL (*SetState)(This,TStateCode vNewState);
	 TStateCode (*GetStateCode)(This);
	 BOOL (*HandleEvent)(This,TEvent vEvent);
Protected
	 Virtual BOOL (*HandleTask)(This,TTask* pvTask);
	 Virtual TStateList* (*GetStateList)(This);
	 TState* (*GetState)(This);
Protected
	 BYTE v[20];
	 TState*  m_pvState;
     TStateCode m_vState;
	 TStateList *m_pStateList;
Private
	 BYTE  m_byPeriod;
	 BYTE  m_byStateProc;
	 BYTE  m_byBoxID;
	 SINT  m_chProcName[DEV_JOB_MAX_PNME];
	 SMESSAGE m_nsMessage;
	 DWORD m_dwAmoutQuant;
	 CMTimer m_nATmr[4];
	 DWORD m_dwTM[4];
	 BYTE m_byAutoState;
	 BYTE V0,V1;
	 DWORD m_dwAutoTime;
	 DECLARE_IMPLEMENT
}
DECLARE_DEFINITION(CCyclicSystem)
#endif
```

#### bnrdbout.h
```c
/********************************************************************
 * COPYRIGHT -- Kontora
 ********************************************************************
 * Program: bnrmain
 * File: bnraninput.h
 * Author: Abramenya
 * Created: January 19, 2009
 *******************************************************************/

#ifndef __DEBUGOUTPUT_H__
#define __DEBUGOUTPUT_H__
#ifdef WIN32
#define DEB_CSensor
#define DEB_CSmartSensor
#define DEB_CDigitalSensor
//#define DEB_CIdleSensor
//#define DEB_CProcManager
#define DEB_CDirectionModule
//#define DEB_CCyclicSystem
#define DEB_CMain
#define DEB_CAdmin
#define DEB_CKpModule
//#define DEB_CMsModule
#define DEB_C101Module
#define DEB_CGsmModule
#define DEB_CTeleSensor
#define DEB_CComServer
#define DEB_CComVS0
#define DEB_CComVS1
#define DEB_CFreq
#define DEB_CStGate
#define DEB_CPunit
#define DEB_CLevel
#define DEB_CObsSys
#define DEB_CMsModule
//#define DEB_CTcpServer
#define DEB_CTeleSignal
#define DEB_CTeleControl
#define DEB_CTeleInd
//#define DEB_CProcManager
#define DEB_CSystem
//#define DEB_CAnIOSlot
//#define DEB_CDgIOSlot
//#define DEB_CAnalogPin
//#define DEB_CDigitalPin
#define DEB_CObserveModule
//#define DEB_CTcpDriver
//#define DEB_CComDriver
//#define DEB_CTcpServer
//#define DEB_CComServer
//#define DEB_CPin
#else
//#define DEB_C101Module
//#define DEB_CComServer
#endif

#endif
```

#### bnrdebug.h
```c
#ifndef DEBUG_H
#define DEBUG_H
#include "typedefs.h"
#include "bnrpob.h"
int  OutFrame(int, BYTE *);
void Info (char *,...);
#endif
```

#### bnrdigsensor.h
```c
/********************************************************************
 * COPYRIGHT -- Kontora
 ********************************************************************
 * Program: bnrmain
 * File: bnraninput.h
 * Author: Abramenya
 * Created: January 19, 2009
 *******************************************************************/

#ifndef __DIGITALSENSOR_H__
#define __DIGITALSENSOR_H__
#include "typedefs.h"
#include "bnrsensr.h"
#if MYSYSTEM_ID != 5
Class CDigitalSensor
{
	 void (*CCDigitalSensor)(This);
	 void (*DCDigitalSensor)(This);
Private
     void (*EventGen)(This);
     void (*SetRemOut)(This,BYTE byNumber,UINT Value);
	 void (*SetPulce)(This,BYTE byNumber,UINT wValue,UINT wTime);
	 void (*PulceGen)(This);
     Virtual void (*InitSensor)(This,SSWITCHTABLE *pSTable);
     Virtual void (*EventHandler)(This,SMESSAGE*);
     Virtual void (*PreProc)(This);
     Virtual void (*Processing)(This);
     Virtual void (*PostProc)(This);
	 Virtual void (*RunAutomat)(This);
Public
     //DWORD m_dwInState;
     //DWORD m_dwOutState;
	 UINT m_nCurrValue[32];
	 UINT m_nPulceTime[32];
	 //BYTE m_byNumber;
     BOOL m_blPulceGo[32];
Private
	 DECLARE_IMPLEMENT_BASE(CSensor)
}
DECLARE_DEFINITION(CDigitalSensor)
#endif
#endif
```

#### bnrdirmodule.h
```c
/********************************************************************
 * COPYRIGHT -- Kontora
 ********************************************************************
 * Program: bnrmain
 * File: bnraninput.h
 * Author: Abramenya
 * Created: January 19, 2009
 *******************************************************************/

#ifndef __OBSERVEMODULE_H__
#define __OBSERVEMODULE_H__
#include "typedefs.h"
#if MYSYSTEM_ID != 5
#include "bnrmessage.h"
#include "bnrsmartsensor.h"
#include "bnridlesensor.h"
#include "bnrdigsensor.h"
#include "bnrcomputer.h"
#include "bnradmin.h"
#include "bnroutgate.h"
#include "bnrflash.h"
#include "bnringate.h"
Class CDirectionModule
{
	void (*CCDirectionModule)(This);
	void (*DCDirectionModule)(This);
Public
	void (*Init)(This,SDIRTABLE *pDirect,CMFlash *pFlash);
    void (*ObserveProc)(This);
	WORD (*GetInOutData)(This,SMESSAGE*);
	void (*SwitchSensor)(This,CSensor *pSensor,SSWITCHTABLE *pSwitchTable);
	void (*SwitchDigitalSensor)(This,CSensor *pSensor,SSWITCHTABLE *pSwitchTable);
	void (*ConnectSensor)(This,CSensor *pSensor,SSWITCHTABLE *pSwitchTable);
	void (*ConnectToComputer)(This,CComputer *pComputer);
	void (*EnableGetData)(This,BOOL);
	void (*ConnectToAdmin)(This,CAdmin*);
	BOOL (*EventHandler)(This,SMESSAGE *pMsg);
	void (*SendMessage)(This,SMESSAGE *pMsg);
	void (*WordXCHG)(This,SMESSAGE *pMsg);
	WORD (*GetXWData)(This,SMESSAGE *pMsg);
	WORD (*GetDigMcData)(This,SMESSAGE *pMsg);
	void (*GetDirMode)(This,SMESSAGE *pMsg);
	void (*SetDirMode)(This,SMESSAGE *pMsg);
	DWORD (*GetDwordParam)(This,BYTE *pbyParam);
	WORD (*GetWordParam)(This,BYTE *pbyParam);
	void (*AddDword)(This,WORD *pwLen,BYTE *byMsg,BYTE *byParam);
	void (*AddWord)(This,WORD *pwLen,BYTE *byMsg,BYTE *byParam);
	void (*SetInputGate)(This,SINPUTGATE *pING);
	BOOL (*Serialize)(This,BOOL blDir);
	BOOL (*SaveContenst)(This);
    BOOL (*LoadContenst)(This);
	void (*SetCurentTank)(This,BYTE byTank);
	void (*SaveTable)(This,SCONTENSTTABLE *psTable);
    void (*LoadTable)(This,SCONTENSTTABLE *psTable);
Private
    CMFlash *m_pFlash;
    CAdmin *m_pAdmin;
	CMTimer m_pStatSnsTmr;
    CComputer *m_pComputer;
	CInputGate m_nInpGate[32];
	PVOID m_pvInGate;
	PVOID m_pvOutGate;
	WORD m_wSensorMode;
	WORD m_wLayerMode;
	BYTE m_byAmInpGate;
	BYTE m_byTypeTest;
	BYTE m_byStatSnsConn;
	BYTE m_byDirectionID;
	BYTE m_byDirectionCode;
	BYTE m_bySystemID;
	BYTE m_byAmSwitching;
	BYTE m_byDefSett;
	BOOL m_blGetData;
	BOOL m_blArmState;
	CSensor **m_pSensor;
	SDIRTABLE *m_pDirTable;
	SCONTENSTTABLE m_nST,m_nCT;
	DECLARE_IMPLEMENT
}
DECLARE_DEFINITION(CDirectionModule)
#endif
#endif
```

#### bnrflash.h
```c
/********************************************************************
 * COPYRIGHT -- Kontora
 ********************************************************************
 * Program: bnrmain
 * File: bnraninput.h
 * Author: Abramenya
 * Created: January 19, 2009
 *******************************************************************/

#ifndef __MFLASH_H__
#define __MFLASH_H__
#include "typedefs.h"
#include "bnrmessage.h"
#ifndef WIN32
 #include <DM_Lib.h>
 #include <dataobj.h>
#else
/* Datatypes and datatypes of function blocks */
#define doERR_MODULNOTFOUND 0
typedef struct DatObjInfo
{
	/* VAR_INPUT (analog) */
	unsigned long pName;
	/* VAR_OUTPUT (analog) */
	unsigned short status;
	unsigned long ident;
	unsigned long pDatObjMem;
	unsigned long len;
	unsigned char MemType;
	unsigned long Option;
	BOOL ChangeDate;
	/* VAR_INPUT (digital) */
	BOOL enable;
} DatObjInfo_typ;
typedef struct DatObjRead
{
	/* VAR_INPUT (analog) */
	unsigned long ident;
	unsigned long Offset;
	unsigned long pDestination;
	unsigned long len;
	/* VAR_OUTPUT (analog) */
	unsigned short status;
	/* VAR_INPUT (digital) */
	BOOL enable;
} DatObjRead_typ;
typedef struct DMxstore
{
	/* VAR_INPUT (analog) */
	unsigned char block_no;
	unsigned long name;
	unsigned long data;
	unsigned long size;
	unsigned long ident;
	/* VAR_OUTPUT (analog) */
	unsigned short status;
	/* VAR_INPUT (digital) */
	BOOL enable;
} DMxstore_typ;

typedef struct DMstore
{
	/* VAR_INPUT (analog) */
	unsigned long name;
	unsigned long data;
	unsigned long size;
	unsigned long ident;
	/* VAR_OUTPUT (analog) */
	unsigned short status;
	/* VAR_INPUT (digital) */
	BOOL enable;
} DMstore_typ;

typedef struct DMxfree
{
	/* VAR_INPUT (analog) */
	unsigned char block_no;
	/* VAR_OUTPUT (analog) */
	unsigned long size;
	unsigned short status;
	/* VAR_INPUT (digital) */
	BOOL enable;
} DMxfree_typ;

typedef struct DMfree
{
	/* VAR_OUTPUT (analog) */
	unsigned long size;
	unsigned short status;
	/* VAR_INPUT (digital) */
	BOOL enable;
} DMfree_typ;

typedef struct DMxclear
{
	/* VAR_INPUT (analog) */
	unsigned char block_no;
	/* VAR_OUTPUT (analog) */
	unsigned short status;
	/* VAR_INPUT (digital) */
	BOOL enable;
} DMxclear_typ;

typedef struct DMclear
{
	/* VAR_OUTPUT (analog) */
	unsigned short status;
	/* VAR_INPUT (digital) */
	BOOL enable;
} DMclear_typ;
/* Prototyping of functions and function blocks */
void DMxstore(struct DMxstore* inst);
void DMstore(struct DMstore* inst);
void DMxfree(struct DMxfree* inst);
void DMfree(struct DMfree* inst);
void DMxclear(struct DMxclear* inst);
void DMclear(struct DMclear* inst);
#endif
Class CMFlash
{
	 void (*CCMFlash)(This);
	 void (*DCMFlash)(This);
Public
     BOOL (*WriteFlash)(This,BYTE *pbyBuff,WORD wLen);
     BOOL (*WriteFlashRem)(This,BYTE *pbyBuff,WORD wLen);
     BOOL (*ReadFlash)(This,BYTE *pbyBuff,WORD wLen);
	 BOOL (*CompareMemory)(This,BYTE *bySrc,WORD wLen);
	 INT  (*Free)(This);
	 BOOL (*ClearFlash)(This);
Private
     char m_chName[30];
     BYTE m_byFirstBlock;
     BYTE m_byAmBlock;
	 DMfree_typ  DM_free;
     DMstore_typ DM_store;
     DMclear_typ DM_clear;
	 DatObjRead_typ DORead;
     DatObjInfo_typ DOInfo;
  	 DECLARE_IMPLEMENT
}
DECLARE_DEFINITION(CMFlash)
#endif
```

#### bnrhardpin.h
```c
/********************************************************************
 * COPYRIGHT -- Kontora
 ********************************************************************
 * Program: bnrmain
 * File: bnraninput.h
 * Author: Abramenya
 * Created: January 19, 2009
 *******************************************************************/

#ifndef __HARDPIN_H__
#define __HARDPIN_H__
#include "typedefs.h"
#include "bnrmessage.h"
#include "bnrpin.h"
//Analog Pin
Class CAnalogPin
{
	 void (*CCAnalogPin)(This);
	 void (*DCAnalogPin)(This);
Public
	 Virtual void (*InitPin)(This,PVOID);
     Virtual void (*SetPin)(This,SPIN*);
	 Virtual void (*GetPin)(This,SPIN*);
	 Virtual PVOID (*GetAddrPin)(This);
	 Virtual PVOID (*GetAddrAlmStatePin)(This);
Private
     UINT *m_vpHardPin;
	 DECLARE_IMPLEMENT_BASE(CPin)
}
DECLARE_DEFINITION(CAnalogPin)
//Digital Pin
Class CDigitalPin
{
	 void (*CCDigitalPin)(This);
	 void (*DCDigitalPin)(This);
Public
	 Virtual void (*InitPin)(This,PVOID);
	 Virtual void (*SetPin)(This,SPIN*);
	 Virtual void (*GetPin)(This,SPIN*);
	 Virtual PVOID (*GetAddrPin)(This);
	 Virtual PVOID (*GetAddrAlmStatePin)(This);
Private
     BOOL *m_vpHardPin;
	 DECLARE_IMPLEMENT_BASE(CPin)
}
DECLARE_DEFINITION(CDigitalPin)
//Counter Pin
Class CDCounterPin
{
	void (*CCDCounterPin)(This);
	void (*DCDCounterPin)(This);
Public
	Virtual void (*InitPin)(This,PVOID);
	Virtual void (*SetPin)(This,SPIN*);
	Virtual void (*GetPin)(This,SPIN*);
	Virtual PVOID (*GetAddrPin)(This);
	Virtual PVOID (*GetAddrAlmStatePin)(This);
Private
	UINT *m_vpHardPin;
	DECLARE_IMPLEMENT_BASE(CPin)
}
DECLARE_DEFINITION(CDCounterPin)
//Temperature Pin
Class CTemperaturePin
{
	void (*CCTemperaturePin)(This);
	void (*DCTemperaturePin)(This);
Public
	Virtual void (*InitPin)(This,PVOID);
	Virtual void (*SetPin)(This,SPIN*);
	Virtual void (*GetPin)(This,SPIN*);
	Virtual PVOID (*GetAddrPin)(This);
	Virtual PVOID (*GetAddrAlmStatePin)(This);
Private
	UINT *m_vpHardPin;
	DECLARE_IMPLEMENT_BASE(CPin)
}
DECLARE_DEFINITION(CTemperaturePin)
#endif
```

#### bnrhconfig.h
```c
/********************************************************************
 * COPYRIGHT -- Kontora
 ********************************************************************
 * Program: bnrmain
 * File: bnrconfig.h
 * Author: Abramenya
 * Created: February 04, 2009
 *******************************************************************/
#ifndef __HARDCONFIG_H__
#define __HARDCONFIG_H__
#ifndef WIN32
#include <bur/plctypes.h>
#endif
#include "typedefs.h"
#include "bnrmessage.h"
void InitHardValue(void);
#endif
```

#### bnridlesensor.h
```c
/********************************************************************
 * COPYRIGHT -- Kontora
 ********************************************************************
 * Program: bnrmain
 * File: bnraninput.h
 * Author: Abramenya
 * Created: January 19, 2009
 *******************************************************************/

#ifndef __IDLESENSOR_H__
#define __IDLESENSOR_H__
#include "typedefs.h"
#if MYSYSTEM_ID != 5
#include "bnrsensr.h"
Class CIdleSensor
{
	 void (*CCIdleSensor)(This);
	 void (*DCIdleSensor)(This);
Public
	 void (*SetMode)(This,USINT);
	 void (*SetState)(This,BOOL);
	 BOOL (*GetState)(This);
Public
	 Virtual void (*InitSensor)(This,PVOID pParam);
     Virtual void (*EventHandler)(This,SMESSAGE*);
     Virtual void (*PreProc)(This);
     Virtual void (*Processing)(This);
     Virtual void (*PostProc)(This);
	 Virtual void (*SetInput)(This,SPIN*);
	 Virtual void (*IncInput)(This,INT16 wParam);
	 Virtual void (*SetOutput)(This,BYTE,SPIN*);
	 Virtual void (*CaptureData)(This);
Private
     BOOL m_blIncInput;
     BOOL m_blDecInput;
     WORD m_iInp;
     WORD m_iOut;
     BOOL m_blState;
	 DECLARE_IMPLEMENT_BASE(CSensor)
}
DECLARE_DEFINITION(CIdleSensor)
#endif
#endif
```

#### bnringate.h
```c
/********************************************************************
 * COPYRIGHT -- Kontora
 ********************************************************************
 * Program: bnrmain
 * File: bnraninput.h
 * Author: Abramenya
 * Created: January 19, 2009
 *******************************************************************/

#ifndef __INGATE_H__
#define __INGATE_H__
#include "typedefs.h"
Class CInputGate
{
	 void (*CCInputGate)(This);
	 void (*DCInputGate)(This);
	 void (*Init)(This,BYTE,UINT*,REAL,REAL);
	 UINT (*GetInput)(This);
	 UINT (*GetMInput)(This);
	 UINT (*GetRealInput)(This);
	 UINT (*HiFilter)(This,UINT);
	 void (*SetResistance)(This,REAL rCurrRes);
	 void (*SetInput)(This,UINT nValue);
     void (*FilterEnable)(This,BYTE);
Public
     BYTE m_byID;
	 BOOL m_blFEnable;
	 BOOL m_blHiInput;
	 UINT *m_pInpGate;
	 UINT m_pInpValue;
	 UINT m_pHiFilMask;
	 UINT m_pInpFreeValue;
     REAL m_rBaseRes;
	 REAL m_rCurrRes;
     REAL m_rKoef;
     /*
	 DINT  PressFilter[260];
     INT16 Fnum;
	 DINT  FSumm, I1, I2, I3;
     INT16 Fval;
	 */
	 DECLARE_IMPLEMENT
}
DECLARE_DEFINITION(CInputGate)
#endif
```

#### bnrkp.h
```c
/********************************************************************
 * COPYRIGHT -- Kontora
 ********************************************************************
 * Program: bnrmain
 * File: bnraninput.h
 * Author: Abramenya
 * Created: January 19, 2009
 *******************************************************************/

#ifndef __KPMODULE_H__
#define __KPMODULE_H__
#include "typedefs.h"
#include "bnrcyclicsystem.h"
#include "bnrtelesensor.h"
#include "bnrtelesignal.h"
#include "bnrteleind.h"
#include "bnrtelecontrol.h"
#include "bnrcomputer.h"
#include "bnrflash.h"

Class CKpModule
{
	 void (*CCKpModule)(This);
	 void (*DCKpModule)(This);
Public
     void (*Init)(This,SHARDCOMPUTERTABLE *pPCTable,SSOFTSWITCHTABLE *pKPTable);
     void (*SaveInPin)(This);
	 void (*SaveAlarmPin)(This);
	 BOOL (*SaveSlotState)(This);
     void (*CreateChannels)(This,SDIRTABLE *pDTable);
	 void (*Connect)(This,SINT *pchPhone);
	 void (*Disconnect)(This);
	 void (*DisconnectL2)(This);
	 void (*StartConnect)(This);
	 void (*CheckSlot)(This);
	 BOOL (*Serialize)(This,BOOL blDir);
	 BOOL (*SaveContenst)(This);
     BOOL (*LoadContenst)(This);
	 void (*StartCheck)(This,BYTE byTime,BYTE byObject);
	 void (*StopCheck)(This);
	 void (*SendObserveMsg)(This);
 	 void (*SaveTable)(This,SCONTENSTTABLE *psTable);
     void (*LoadTable)(This,SCONTENSTTABLE *psTable);
     Virtual BOOL (*EventHandler)(This,SMESSAGE *pMsg);
     Virtual void (*CyclicProc)(This);
Public
     CTeleSensor **m_pTeleSensor;
     CComputer *m_pComputer;
	 CMTimer m_nConnTMR,m_nDiscTMR,m_pResetTimer,m_nConnRepTMP,m_nPuCommTMR,m_nSDiscTMR,m_nRepConnTMR;
	 SCONTENSTTABLE m_nST,m_nCT;
	 SHARDCOMPUTERTABLE *m_pPCT;
	 SSOFTSWITCHTABLE   *m_pPST;
	 SKPPARAM *m_pKP;
	 SDIRTABLE *m_pD;
	 CMFlash m_nFlash;
	 CMFlash *m_pFlash;
	 BOOL m_blBufferST;
	 BOOL m_blDiscStart;
	 BOOL m_blIfConnect;
	 BYTE m_byObsTime;
	 BYTE m_byObsObject;
	 BYTE m_byDiscProc;
	 BYTE m_byConnCT;
	 BYTE m_byCallCT;
	 BYTE m_byKpState;
     BYTE m_byKpID;
	 WORD m_wAmChannel,m_wCallTime;
	 DECLARE_IMPLEMENT_BASE(CCyclicSystem)
}
DECLARE_DEFINITION(CKpModule)
#endif
```

#### bnrmain.h
```c
/********************************************************************
 * COPYRIGHT -- Kontora
 ********************************************************************
 * Program: bnrmain
 * File: bnrmain.h
 * Author: Abramenya
 * Created: January 19, 2009
 *******************************************************************/

#include "typedefs.h"
#include "bnrmysystem.h"
#include "bnrprocmanager.h"
#include "bnrdebug.h"
#include "bnrpob.h"
#ifndef WIN32
#include <bur/plctypes.h>
#else
#include "time.h"
#endif
void _INIT bnrmainINIT( void );
void _CYCLIC bnrmainCYCLIC( void );
void SetBoardTime(BYTE *byTime);
void SendSMessage(BYTE byBox,BYTE byFor,BYTE byType);
void SendCommand(BYTE byEvent,SINT *pchCommand);
void SendChar(BYTE byEvent,SINT *pchCommand);
#ifdef WIN32
  DWORD WINAPI CyclicProcess(PVOID);
  void CreateCyclicProc(void);
  void GetSysCommand(void);
  void heapdump( void );
#endif
  void GetCurTime(STIME *pTime);
  void _EXIT bnrmainEXIT( void );
  BOOL CreateSystem(SHARDCOMPUTERTABLE *plConfigTable);
  BOOL CreateProcManager(void/*CSystem *pSystem*/);
  void InitSystem(void);
  void DeleteSystem(void);
#ifndef WIN32
int main(void);
#endif
```
